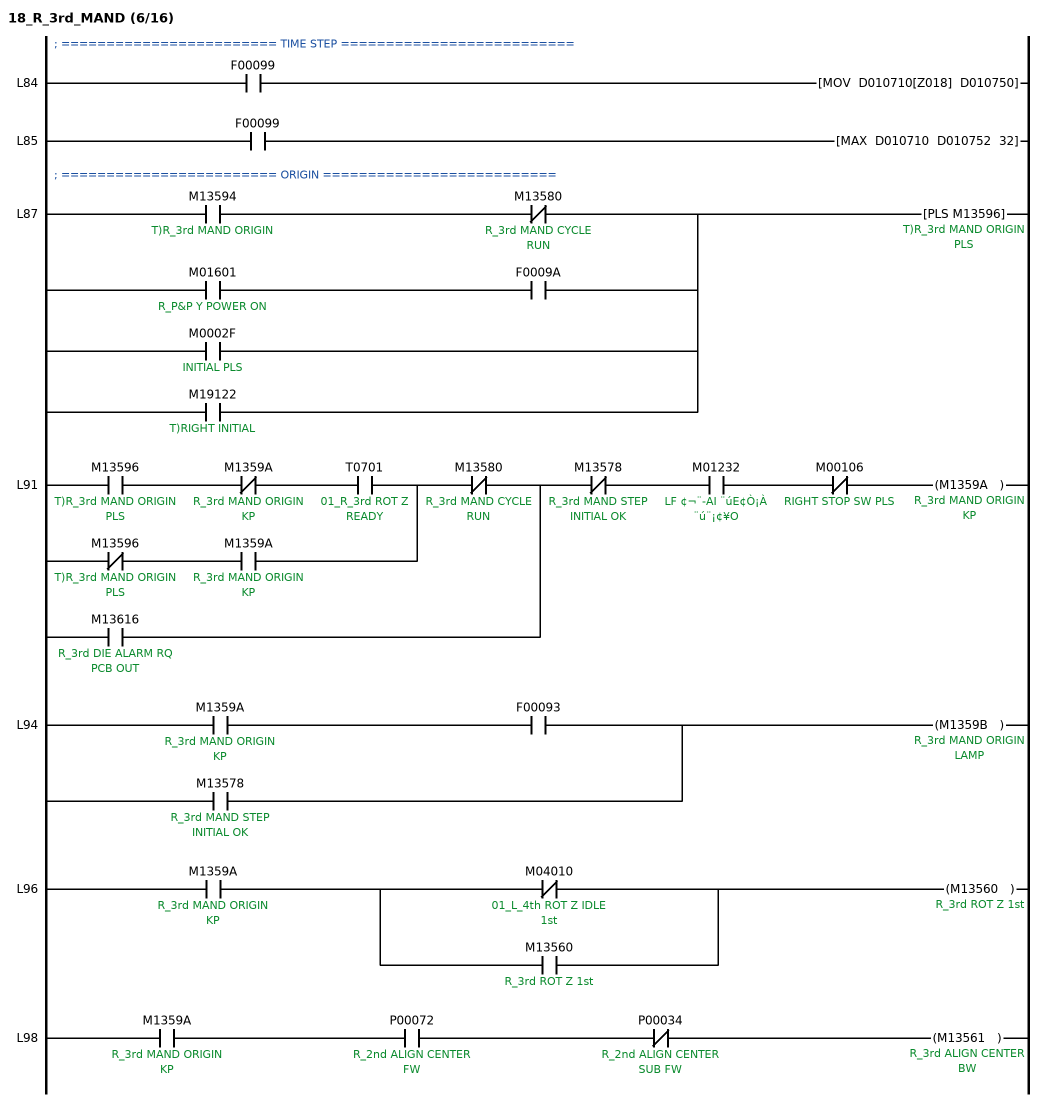
[picture p168: 18_R_3rd_MAND rungs L84-L98]
// ======================== TIME STEP ==========================
; L84
LOAD      F00099
MOV       D010710[Z018] D010750
; L85
LOAD      F00099
MAX       D010710 D010752 32
// ======================== ORIGIN ==========================
; L87
LOAD      M13594	// T)R_3rd MAND ORIGIN
AND NOT   M13580	// R_3rd MAND CYCLE RUN
LOAD      M01601	// R_P&P Y POWER ON
AND       F0009A
OR LOAD
OR        M0002F	// INITIAL PLS
OR        M19122	// T)RIGHT INITIAL
OUTP      M13596	// T)R_3rd MAND ORIGIN PLS
; L91
LOAD      M13596	// T)R_3rd MAND ORIGIN PLS
AND NOT   M1359A	// R_3rd MAND ORIGIN KP
AND       T0701	// 01_R_3rd ROT Z READY
LOAD NOT  M13596	// T)R_3rd MAND ORIGIN PLS
AND       M1359A	// R_3rd MAND ORIGIN KP
OR LOAD
AND NOT   M13580	// R_3rd MAND CYCLE RUN
OR        M13616	// R_3rd DIE ALARM RQ PCB OUT
AND NOT   M13578	// R_3rd MAND STEP INITIAL OK
AND       M01232	// LF ¢¬¨­AI ¨úE¢Ò¡À ¨ú¨¡¢¥O
AND NOT   M00106	// RIGHT STOP SW PLS
OUT       M1359A	// R_3rd MAND ORIGIN KP
; L94
LOAD      M1359A	// R_3rd MAND ORIGIN KP
AND       F00093
OR        M13578	// R_3rd MAND STEP INITIAL OK
OUT       M1359B	// R_3rd MAND ORIGIN LAMP
; L96
LOAD      M1359A	// R_3rd MAND ORIGIN KP
LOAD NOT  M04010	// 01_L_4th ROT Z IDLE 1st
OR        M13560	// R_3rd ROT Z 1st
AND LOAD
OUT       M13560	// R_3rd ROT Z 1st
; L98
LOAD      M1359A	// R_3rd MAND ORIGIN KP
AND       P00072	// R_2nd ALIGN CENTER FW
AND NOT   P00034	// R_2nd ALIGN CENTER SUB FW
OUT       M13561	// R_3rd ALIGN CENTER BW

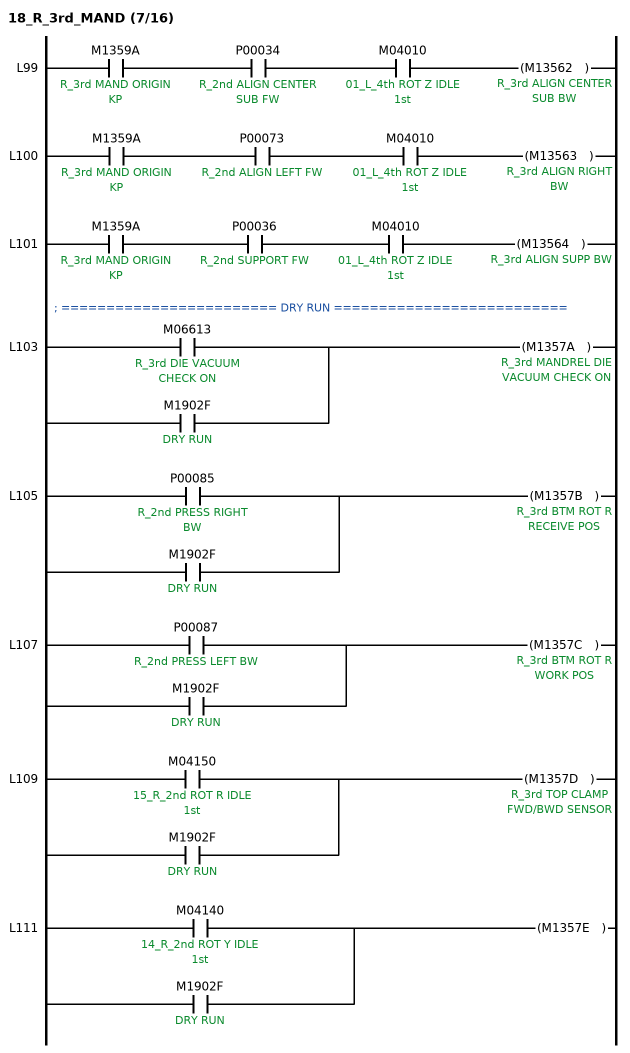
; L99
LOAD      M1359A	// R_3rd MAND ORIGIN KP
AND       P00034	// R_2nd ALIGN CENTER SUB FW
AND       M04010	// 01_L_4th ROT Z IDLE 1st
OUT       M13562	// R_3rd ALIGN CENTER SUB BW
; L100
LOAD      M1359A	// R_3rd MAND ORIGIN KP
AND       P00073	// R_2nd ALIGN LEFT FW
AND       M04010	// 01_L_4th ROT Z IDLE 1st
OUT       M13563	// R_3rd ALIGN RIGHT BW
; L101
LOAD      M1359A	// R_3rd MAND ORIGIN KP
AND       P00036	// R_2nd SUPPORT FW
AND       M04010	// 01_L_4th ROT Z IDLE 1st
OUT       M13564	// R_3rd ALIGN SUPP BW
// ======================== DRY RUN ==========================
; L103
LOAD      M06613	// R_3rd DIE VACUUM CHECK ON
OR        M1902F	// DRY RUN
OUT       M1357A	// R_3rd MANDREL DIE VACUUM CHECK ON
; L105
LOAD      P00085	// R_2nd PRESS RIGHT BW
OR        M1902F	// DRY RUN
OUT       M1357B	// R_3rd BTM ROT R RECEIVE POS
; L107
LOAD      P00087	// R_2nd PRESS LEFT BW
OR        M1902F	// DRY RUN
OUT       M1357C	// R_3rd BTM ROT R WORK POS
; L109
LOAD      M04150	// 15_R_2nd ROT R IDLE 1st
OR        M1902F	// DRY RUN
OUT       M1357D	// R_3rd TOP CLAMP FWD/BWD SENSOR
; L111
LOAD      M04140	// 14_R_2nd ROT Y IDLE 1st
OR        M1902F	// DRY RUN
OUT       M1357E

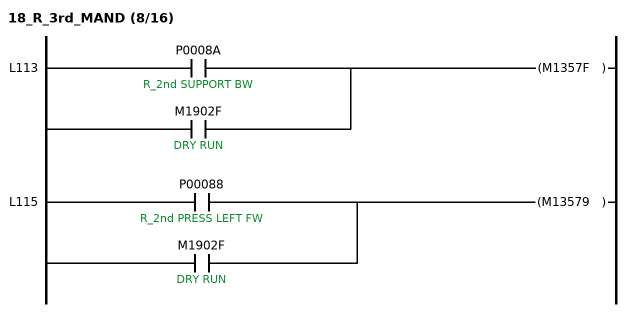
; L113
LOAD      P0008A	// R_2nd SUPPORT BW
OR        M1902F	// DRY RUN
OUT       M1357F
; L115
LOAD      P00088	// R_2nd PRESS LEFT FW
OR        M1902F	// DRY RUN
OUT       M13579

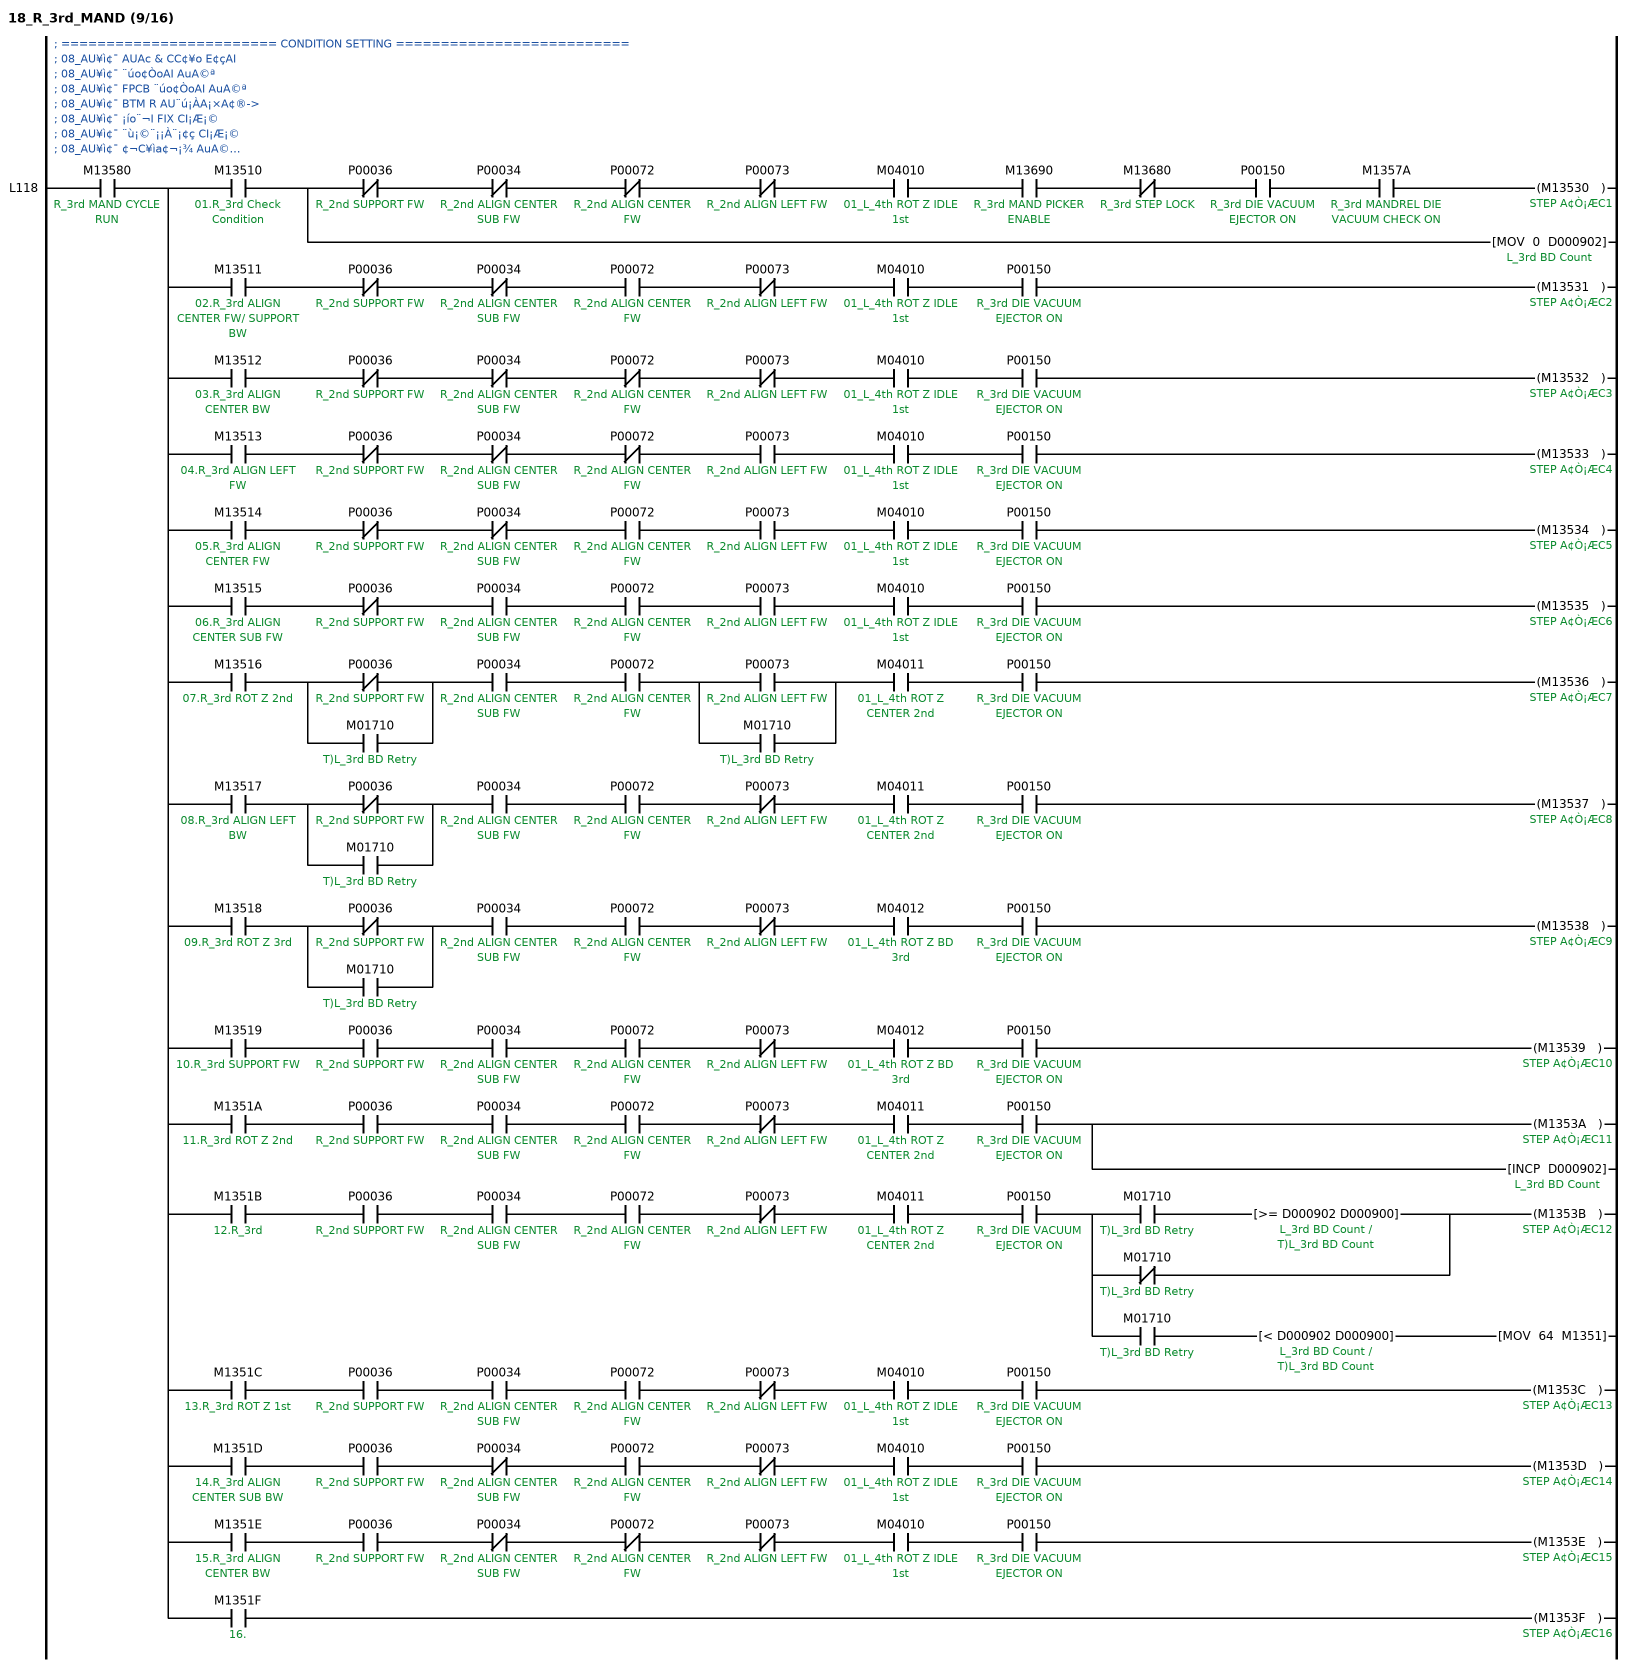
// ======================== CONDITION SETTING ==========================
; L118
LOAD      M13580	// R_3rd MAND CYCLE RUN
MPUSH
AND       M13510	// 01.R_3rd Check Condition
MPUSH
AND NOT   P00036	// R_2nd SUPPORT FW
AND NOT   P00034	// R_2nd ALIGN CENTER SUB FW
AND NOT   P00072	// R_2nd ALIGN CENTER FW
AND NOT   P00073	// R_2nd ALIGN LEFT FW
AND       M04010	// 01_L_4th ROT Z IDLE 1st
AND       M13690	// R_3rd MAND PICKER ENABLE
AND NOT   M13680	// R_3rd STEP LOCK
AND       P00150	// R_3rd DIE VACUUM EJECTOR ON
AND       M1357A	// R_3rd MANDREL DIE VACUUM CHECK ON
OUT       M13530	// STEP A¢Ò¡ÆC1
MPOP
MOV       0 D000902	// L_3rd BD Count
MLOAD
AND       M13511	// 02.R_3rd ALIGN CENTER FW/ SUPPORT BW
AND NOT   P00036	// R_2nd SUPPORT FW
AND NOT   P00034	// R_2nd ALIGN CENTER SUB FW
AND       P00072	// R_2nd ALIGN CENTER FW
AND NOT   P00073	// R_2nd ALIGN LEFT FW
AND       M04010	// 01_L_4th ROT Z IDLE 1st
AND       P00150	// R_3rd DIE VACUUM EJECTOR ON
OUT       M13531	// STEP A¢Ò¡ÆC2
MLOAD
AND       M13512	// 03.R_3rd ALIGN CENTER BW
AND NOT   P00036	// R_2nd SUPPORT FW
AND NOT   P00034	// R_2nd ALIGN CENTER SUB FW
AND NOT   P00072	// R_2nd ALIGN CENTER FW
AND NOT   P00073	// R_2nd ALIGN LEFT FW
AND       M04010	// 01_L_4th ROT Z IDLE 1st
AND       P00150	// R_3rd DIE VACUUM EJECTOR ON
OUT       M13532	// STEP A¢Ò¡ÆC3
MLOAD
AND       M13513	// 04.R_3rd ALIGN LEFT FW
AND NOT   P00036	// R_2nd SUPPORT FW
AND NOT   P00034	// R_2nd ALIGN CENTER SUB FW
AND NOT   P00072	// R_2nd ALIGN CENTER FW
AND       P00073	// R_2nd ALIGN LEFT FW
AND       M04010	// 01_L_4th ROT Z IDLE 1st
AND       P00150	// R_3rd DIE VACUUM EJECTOR ON
OUT       M13533	// STEP A¢Ò¡ÆC4
MLOAD
AND       M13514	// 05.R_3rd ALIGN CENTER FW
AND NOT   P00036	// R_2nd SUPPORT FW
AND NOT   P00034	// R_2nd ALIGN CENTER SUB FW
AND       P00072	// R_2nd ALIGN CENTER FW
AND       P00073	// R_2nd ALIGN LEFT FW
AND       M04010	// 01_L_4th ROT Z IDLE 1st
AND       P00150	// R_3rd DIE VACUUM EJECTOR ON
OUT       M13534	// STEP A¢Ò¡ÆC5
MLOAD
AND       M13515	// 06.R_3rd ALIGN CENTER SUB FW
AND NOT   P00036	// R_2nd SUPPORT FW
AND       P00034	// R_2nd ALIGN CENTER SUB FW
AND       P00072	// R_2nd ALIGN CENTER FW
AND       P00073	// R_2nd ALIGN LEFT FW
AND       M04010	// 01_L_4th ROT Z IDLE 1st
AND       P00150	// R_3rd DIE VACUUM EJECTOR ON
OUT       M13535	// STEP A¢Ò¡ÆC6
MLOAD
AND       M13516	// 07.R_3rd ROT Z 2nd
LOAD NOT  P00036	// R_2nd SUPPORT FW
OR        M01710	// T)L_3rd BD Retry
AND LOAD
AND       P00034	// R_2nd ALIGN CENTER SUB FW
AND       P00072	// R_2nd ALIGN CENTER FW
LOAD      P00073	// R_2nd ALIGN LEFT FW
OR        M01710	// T)L_3rd BD Retry
AND LOAD
AND       M04011	// 01_L_4th ROT Z CENTER 2nd
AND       P00150	// R_3rd DIE VACUUM EJECTOR ON
OUT       M13536	// STEP A¢Ò¡ÆC7
MLOAD
AND       M13517	// 08.R_3rd ALIGN LEFT BW
LOAD NOT  P00036	// R_2nd SUPPORT FW
OR        M01710	// T)L_3rd BD Retry
AND LOAD
AND       P00034	// R_2nd ALIGN CENTER SUB FW
AND       P00072	// R_2nd ALIGN CENTER FW
AND NOT   P00073	// R_2nd ALIGN LEFT FW
AND       M04011	// 01_L_4th ROT Z CENTER 2nd
AND       P00150	// R_3rd DIE VACUUM EJECTOR ON
OUT       M13537	// STEP A¢Ò¡ÆC8
MLOAD
AND       M13518	// 09.R_3rd ROT Z 3rd
LOAD NOT  P00036	// R_2nd SUPPORT FW
OR        M01710	// T)L_3rd BD Retry
AND LOAD
AND       P00034	// R_2nd ALIGN CENTER SUB FW
AND       P00072	// R_2nd ALIGN CENTER FW
AND NOT   P00073	// R_2nd ALIGN LEFT FW
AND       M04012	// 01_L_4th ROT Z BD 3rd
AND       P00150	// R_3rd DIE VACUUM EJECTOR ON
OUT       M13538	// STEP A¢Ò¡ÆC9
MLOAD
AND       M13519	// 10.R_3rd SUPPORT FW
AND       P00036	// R_2nd SUPPORT FW
AND       P00034	// R_2nd ALIGN CENTER SUB FW
AND       P00072	// R_2nd ALIGN CENTER FW
AND NOT   P00073	// R_2nd ALIGN LEFT FW
AND       M04012	// 01_L_4th ROT Z BD 3rd
AND       P00150	// R_3rd DIE VACUUM EJECTOR ON
OUT       M13539	// STEP A¢Ò¡ÆC10
MLOAD
AND       M1351A	// 11.R_3rd ROT Z 2nd
AND       P00036	// R_2nd SUPPORT FW
AND       P00034	// R_2nd ALIGN CENTER SUB FW
AND       P00072	// R_2nd ALIGN CENTER FW
AND NOT   P00073	// R_2nd ALIGN LEFT FW
AND       M04011	// 01_L_4th ROT Z CENTER 2nd
AND       P00150	// R_3rd DIE VACUUM EJECTOR ON
OUT       M1353A	// STEP A¢Ò¡ÆC11
INCP      D000902	// L_3rd BD Count
MLOAD
AND       M1351B	// 12.R_3rd 
AND       P00036	// R_2nd SUPPORT FW
AND       P00034	// R_2nd ALIGN CENTER SUB FW
AND       P00072	// R_2nd ALIGN CENTER FW
AND NOT   P00073	// R_2nd ALIGN LEFT FW
AND       M04011	// 01_L_4th ROT Z CENTER 2nd
AND       P00150	// R_3rd DIE VACUUM EJECTOR ON
MPUSH
LOAD      M01710	// T)L_3rd BD Retry
AND>=     D000902 D000900	// L_3rd BD Count / T)L_3rd BD Count
OR NOT    M01710	// T)L_3rd BD Retry
AND LOAD
OUT       M1353B	// STEP A¢Ò¡ÆC12
MPOP
AND       M01710	// T)L_3rd BD Retry
AND<      D000902 D000900	// L_3rd BD Count / T)L_3rd BD Count
MOV       64 M1351
MLOAD
AND       M1351C	// 13.R_3rd ROT Z 1st
AND       P00036	// R_2nd SUPPORT FW
AND       P00034	// R_2nd ALIGN CENTER SUB FW
AND       P00072	// R_2nd ALIGN CENTER FW
AND NOT   P00073	// R_2nd ALIGN LEFT FW
AND       M04010	// 01_L_4th ROT Z IDLE 1st
AND       P00150	// R_3rd DIE VACUUM EJECTOR ON
OUT       M1353C	// STEP A¢Ò¡ÆC13
MLOAD
AND       M1351D	// 14.R_3rd ALIGN CENTER SUB BW
AND       P00036	// R_2nd SUPPORT FW
AND NOT   P00034	// R_2nd ALIGN CENTER SUB FW
AND       P00072	// R_2nd ALIGN CENTER FW
AND NOT   P00073	// R_2nd ALIGN LEFT FW
AND       M04010	// 01_L_4th ROT Z IDLE 1st
AND       P00150	// R_3rd DIE VACUUM EJECTOR ON
OUT       M1353D	// STEP A¢Ò¡ÆC14
MLOAD
AND       M1351E	// 15.R_3rd ALIGN CENTER BW
AND       P00036	// R_2nd SUPPORT FW
AND NOT   P00034	// R_2nd ALIGN CENTER SUB FW
AND NOT   P00072	// R_2nd ALIGN CENTER FW
AND NOT   P00073	// R_2nd ALIGN LEFT FW
AND       M04010	// 01_L_4th ROT Z IDLE 1st
AND       P00150	// R_3rd DIE VACUUM EJECTOR ON
OUT       M1353E	// STEP A¢Ò¡ÆC15
MPOP
AND       M1351F	// 16.
OUT       M1353F	// STEP A¢Ò¡ÆC16
// output comment: 08_AU¥ì¢¯ AUAc & CC¢¥o E¢çAI
// output comment: 08_AU¥ì¢¯ ¨úo¢ÒoAI AuA©ª
// output comment: 08_AU¥ì¢¯ FPCB ¨úo¢ÒoAI AuA©ª
// output comment: 08_AU¥ì¢¯ BTM R AU¨ú¡ÀA¡×A¢®->
// output comment: 08_AU¥ì¢¯ ¡ío¨¬I FIX CI¡Æ¡©
// output comment: 08_AU¥ì¢¯ ¨ù¡©¨¡¡À¨¡¢ç CI¡Æ¡©
// output comment: 08_AU¥ì¢¯ ¢¬C¥ìa¢¬¡¾ AuA©ª
// output comment: 08_AU¥ì¢¯ ¢¬C¥ìa¢¬¡¾ E¢¬Au
// output comment: 08_AU¥ì¢¯ ¢¬C¥ìa¢¬¡¾ ¨¬©ö¡¾I

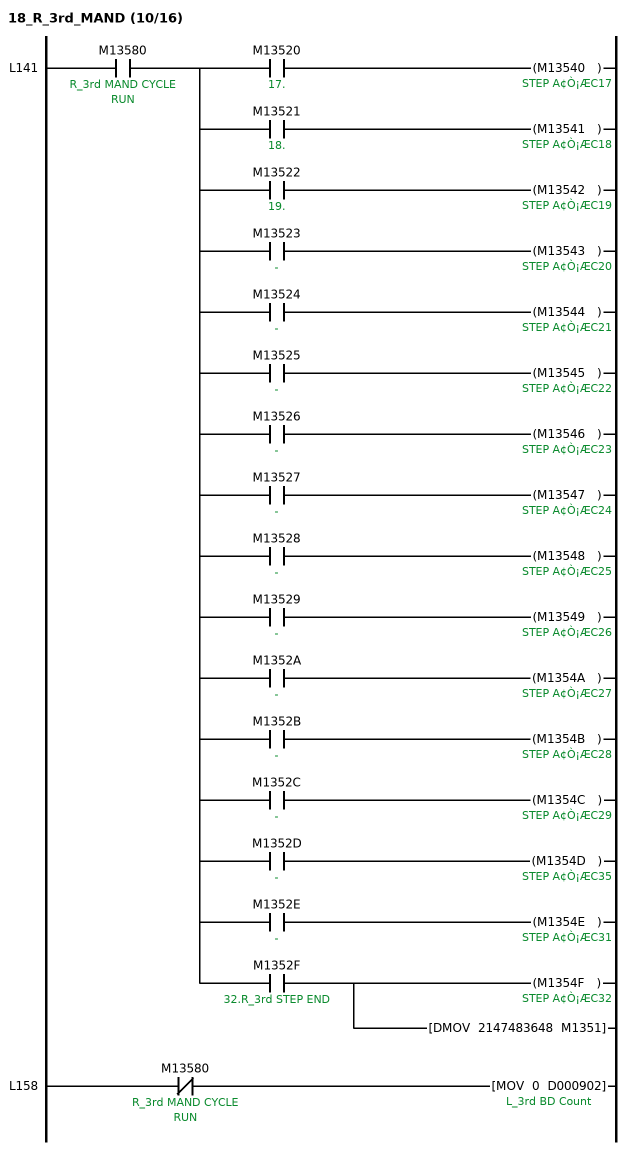
; L141
LOAD      M13580	// R_3rd MAND CYCLE RUN
MPUSH
AND       M13520	// 17.
OUT       M13540	// STEP A¢Ò¡ÆC17
MLOAD
AND       M13521	// 18.
OUT       M13541	// STEP A¢Ò¡ÆC18
MLOAD
AND       M13522	// 19.
OUT       M13542	// STEP A¢Ò¡ÆC19
MLOAD
AND       M13523	// -
OUT       M13543	// STEP A¢Ò¡ÆC20
MLOAD
AND       M13524	// -
OUT       M13544	// STEP A¢Ò¡ÆC21
MLOAD
AND       M13525	// -
OUT       M13545	// STEP A¢Ò¡ÆC22
MLOAD
AND       M13526	// -
OUT       M13546	// STEP A¢Ò¡ÆC23
MLOAD
AND       M13527	// -
OUT       M13547	// STEP A¢Ò¡ÆC24
MLOAD
AND       M13528	// -
OUT       M13548	// STEP A¢Ò¡ÆC25
MLOAD
AND       M13529	// -
OUT       M13549	// STEP A¢Ò¡ÆC26
MLOAD
AND       M1352A	// -
OUT       M1354A	// STEP A¢Ò¡ÆC27
MLOAD
AND       M1352B	// -
OUT       M1354B	// STEP A¢Ò¡ÆC28
MLOAD
AND       M1352C	// -
OUT       M1354C	// STEP A¢Ò¡ÆC29
MLOAD
AND       M1352D	// -
OUT       M1354D	// STEP A¢Ò¡ÆC35
MLOAD
AND       M1352E	// -
OUT       M1354E	// STEP A¢Ò¡ÆC31
MPOP
AND       M1352F	// 32.R_3rd STEP END
OUT       M1354F	// STEP A¢Ò¡ÆC32
DMOV      2147483648 M1351
; L158
LOAD NOT  M13580	// R_3rd MAND CYCLE RUN
MOV       0 D000902	// L_3rd BD Count

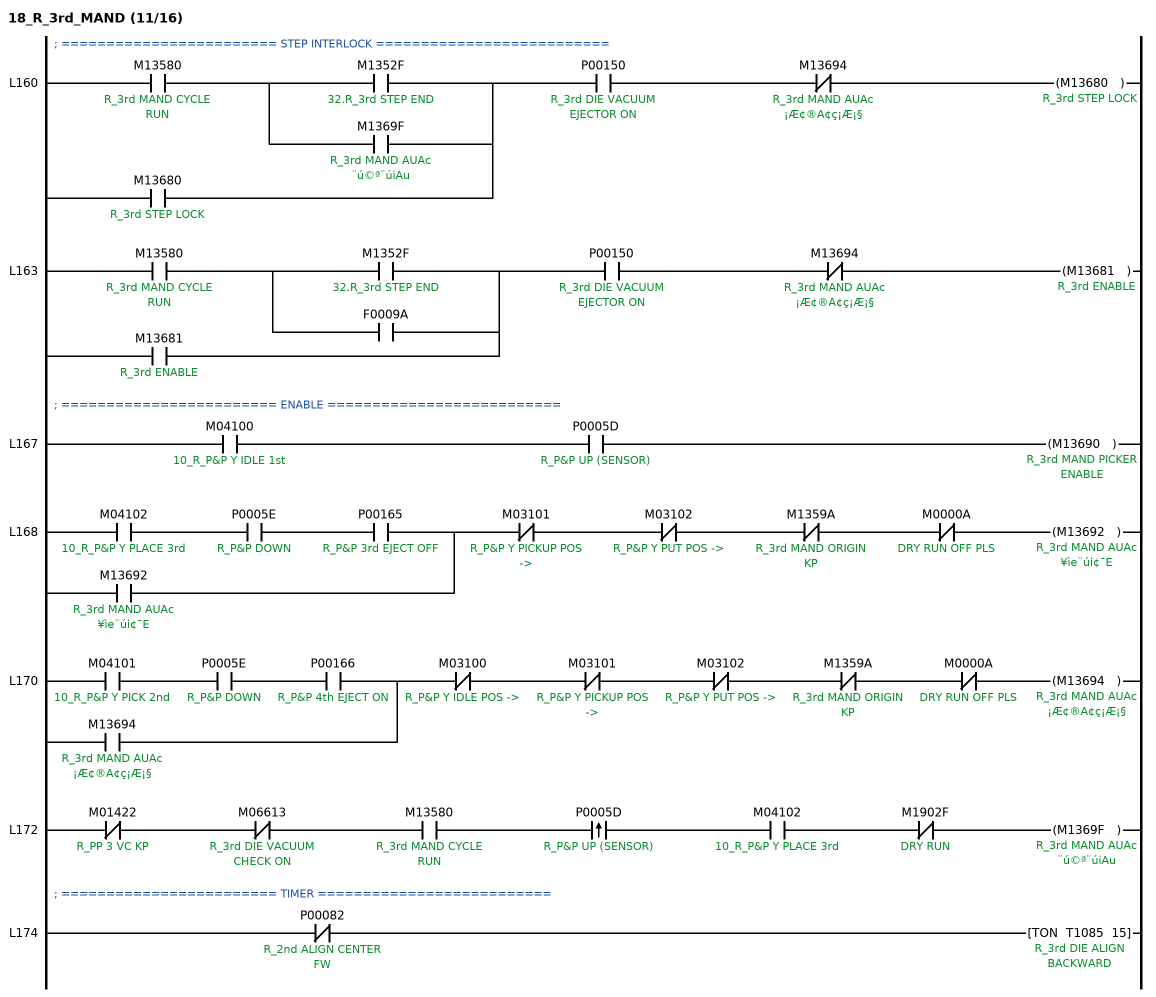
// ======================== STEP INTERLOCK ==========================
; L160
LOAD      M13580	// R_3rd MAND CYCLE RUN
LOAD      M1352F	// 32.R_3rd STEP END
OR        M1369F	// R_3rd MAND AUAc ¨ú©ª¨úiAu
AND LOAD
OR        M13680	// R_3rd STEP LOCK
AND       P00150	// R_3rd DIE VACUUM EJECTOR ON
AND NOT   M13694	// R_3rd MAND AUAc ¡Æ¢®A¢ç¡Æ¡§
OUT       M13680	// R_3rd STEP LOCK
; L163
LOAD      M13580	// R_3rd MAND CYCLE RUN
LOAD      M1352F	// 32.R_3rd STEP END
OR        F0009A
AND LOAD
OR        M13681	// R_3rd ENABLE
AND       P00150	// R_3rd DIE VACUUM EJECTOR ON
AND NOT   M13694	// R_3rd MAND AUAc ¡Æ¢®A¢ç¡Æ¡§
OUT       M13681	// R_3rd ENABLE
// ======================== ENABLE ==========================
; L167
LOAD      M04100	// 10_R_P&P Y IDLE 1st
AND       P0005D	// R_P&P UP (SENSOR)
OUT       M13690	// R_3rd MAND PICKER ENABLE
; L168
LOAD      M04102	// 10_R_P&P Y PLACE 3rd
AND       P0005E	// R_P&P DOWN
AND       P00165	// R_P&P 3rd EJECT OFF
OR        M13692	// R_3rd MAND AUAc ¥ìe¨úi¢¯E
AND NOT   M03101	// R_P&P Y PICKUP POS ->
AND NOT   M03102	// R_P&P Y PUT POS ->
AND NOT   M1359A	// R_3rd MAND ORIGIN KP
AND NOT   M0000A	// DRY RUN OFF PLS
OUT       M13692	// R_3rd MAND AUAc ¥ìe¨úi¢¯E
; L170
LOAD      M04101	// 10_R_P&P Y PICK 2nd
AND       P0005E	// R_P&P DOWN
AND       P00166	// R_P&P 4th EJECT ON
OR        M13694	// R_3rd MAND AUAc ¡Æ¢®A¢ç¡Æ¡§
AND NOT   M03100	// R_P&P Y IDLE POS ->
AND NOT   M03101	// R_P&P Y PICKUP POS ->
AND NOT   M03102	// R_P&P Y PUT POS ->
AND NOT   M1359A	// R_3rd MAND ORIGIN KP
AND NOT   M0000A	// DRY RUN OFF PLS
OUT       M13694	// R_3rd MAND AUAc ¡Æ¢®A¢ç¡Æ¡§
; L172
LOAD NOT  M01422	// R_PP 3 VC KP
AND NOT   M06613	// R_3rd DIE VACUUM CHECK ON
AND       M13580	// R_3rd MAND CYCLE RUN
ANDP      P0005D	// R_P&P UP (SENSOR)
AND       M04102	// 10_R_P&P Y PLACE 3rd
AND NOT   M1902F	// DRY RUN
OUT       M1369F	// R_3rd MAND AUAc ¨ú©ª¨úiAu
// ======================== TIMER ==========================
; L174
LOAD NOT  P00082	// R_2nd ALIGN CENTER FW
TON       T1085 15	// R_3rd DIE ALIGN BACKWARD

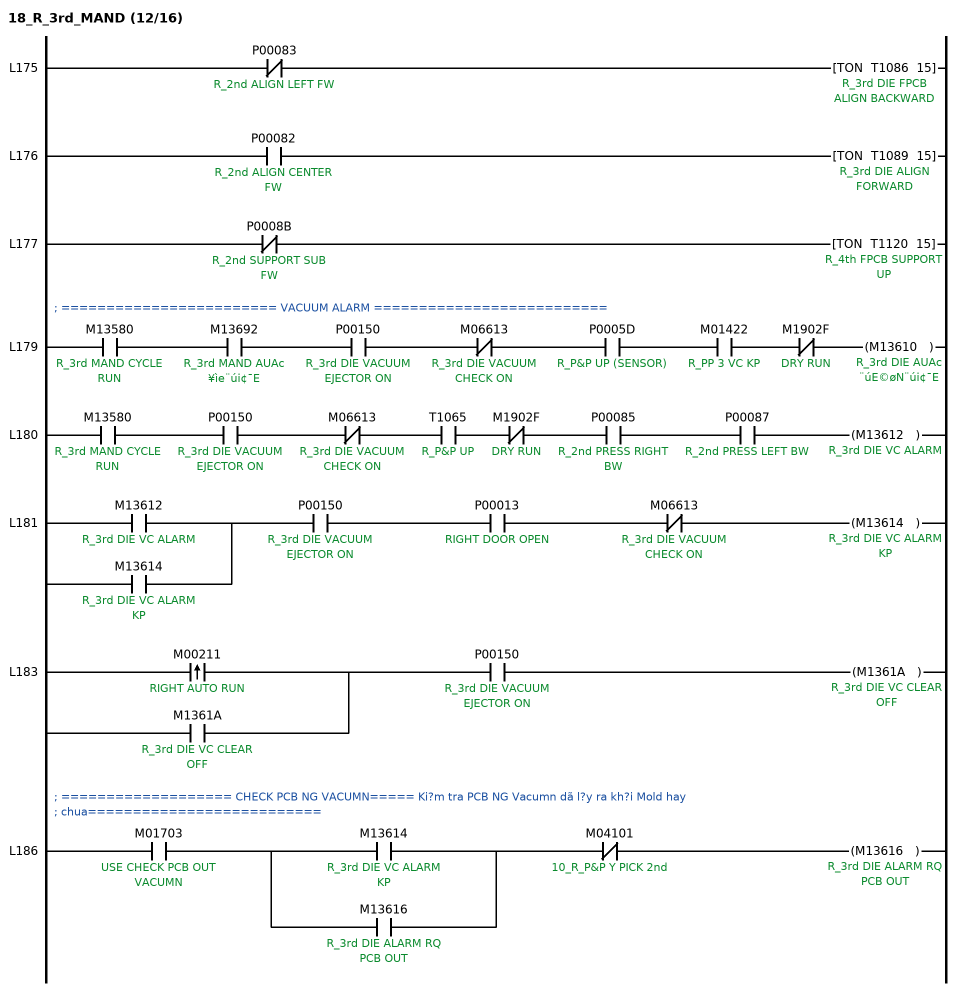
; L175
LOAD NOT  P00083	// R_2nd ALIGN LEFT FW
TON       T1086 15	// R_3rd DIE FPCB ALIGN BACKWARD
; L176
LOAD      P00082	// R_2nd ALIGN CENTER FW
TON       T1089 15	// R_3rd DIE ALIGN FORWARD
; L177
LOAD NOT  P0008B	// R_2nd SUPPORT SUB FW
TON       T1120 15	// R_4th FPCB SUPPORT UP
// ======================== VACUUM ALARM ==========================
; L179
LOAD      M13580	// R_3rd MAND CYCLE RUN
AND       M13692	// R_3rd MAND AUAc ¥ìe¨úi¢¯E
AND       P00150	// R_3rd DIE VACUUM EJECTOR ON
AND NOT   M06613	// R_3rd DIE VACUUM CHECK ON
AND       P0005D	// R_P&P UP (SENSOR)
AND       M01422	// R_PP 3 VC KP
AND NOT   M1902F	// DRY RUN
OUT       M13610	// R_3rd DIE AUAc ¨úE©øN¨úi¢¯E
; L180
LOAD      M13580	// R_3rd MAND CYCLE RUN
AND       P00150	// R_3rd DIE VACUUM EJECTOR ON
AND NOT   M06613	// R_3rd DIE VACUUM CHECK ON
AND       T1065	// R_P&P UP
AND NOT   M1902F	// DRY RUN
AND       P00085	// R_2nd PRESS RIGHT BW
AND       P00087	// R_2nd PRESS LEFT BW
OUT       M13612	// R_3rd DIE VC ALARM
; L181
LOAD      M13612	// R_3rd DIE VC ALARM
OR        M13614	// R_3rd DIE VC ALARM KP
AND       P00150	// R_3rd DIE VACUUM EJECTOR ON
AND       P00013	// RIGHT DOOR OPEN
AND NOT   M06613	// R_3rd DIE VACUUM CHECK ON
OUT       M13614	// R_3rd DIE VC ALARM KP
; L183
LOADP     M00211	// RIGHT AUTO RUN
OR        M1361A	// R_3rd DIE VC CLEAR OFF
AND       P00150	// R_3rd DIE VACUUM EJECTOR ON
OUT       M1361A	// R_3rd DIE VC CLEAR OFF
// =================== CHECK PCB NG VACUMN===== Ki?m tra PCB NG Vacumn dã l?y ra kh?i Mold hay chua==========================
; L186
LOAD      M01703	// USE CHECK PCB OUT VACUMN
LOAD      M13614	// R_3rd DIE VC ALARM KP
OR        M13616	// R_3rd DIE ALARM RQ PCB OUT
AND LOAD
AND NOT   M04101	// 10_R_P&P Y PICK 2nd
OUT       M13616	// R_3rd DIE ALARM RQ PCB OUT

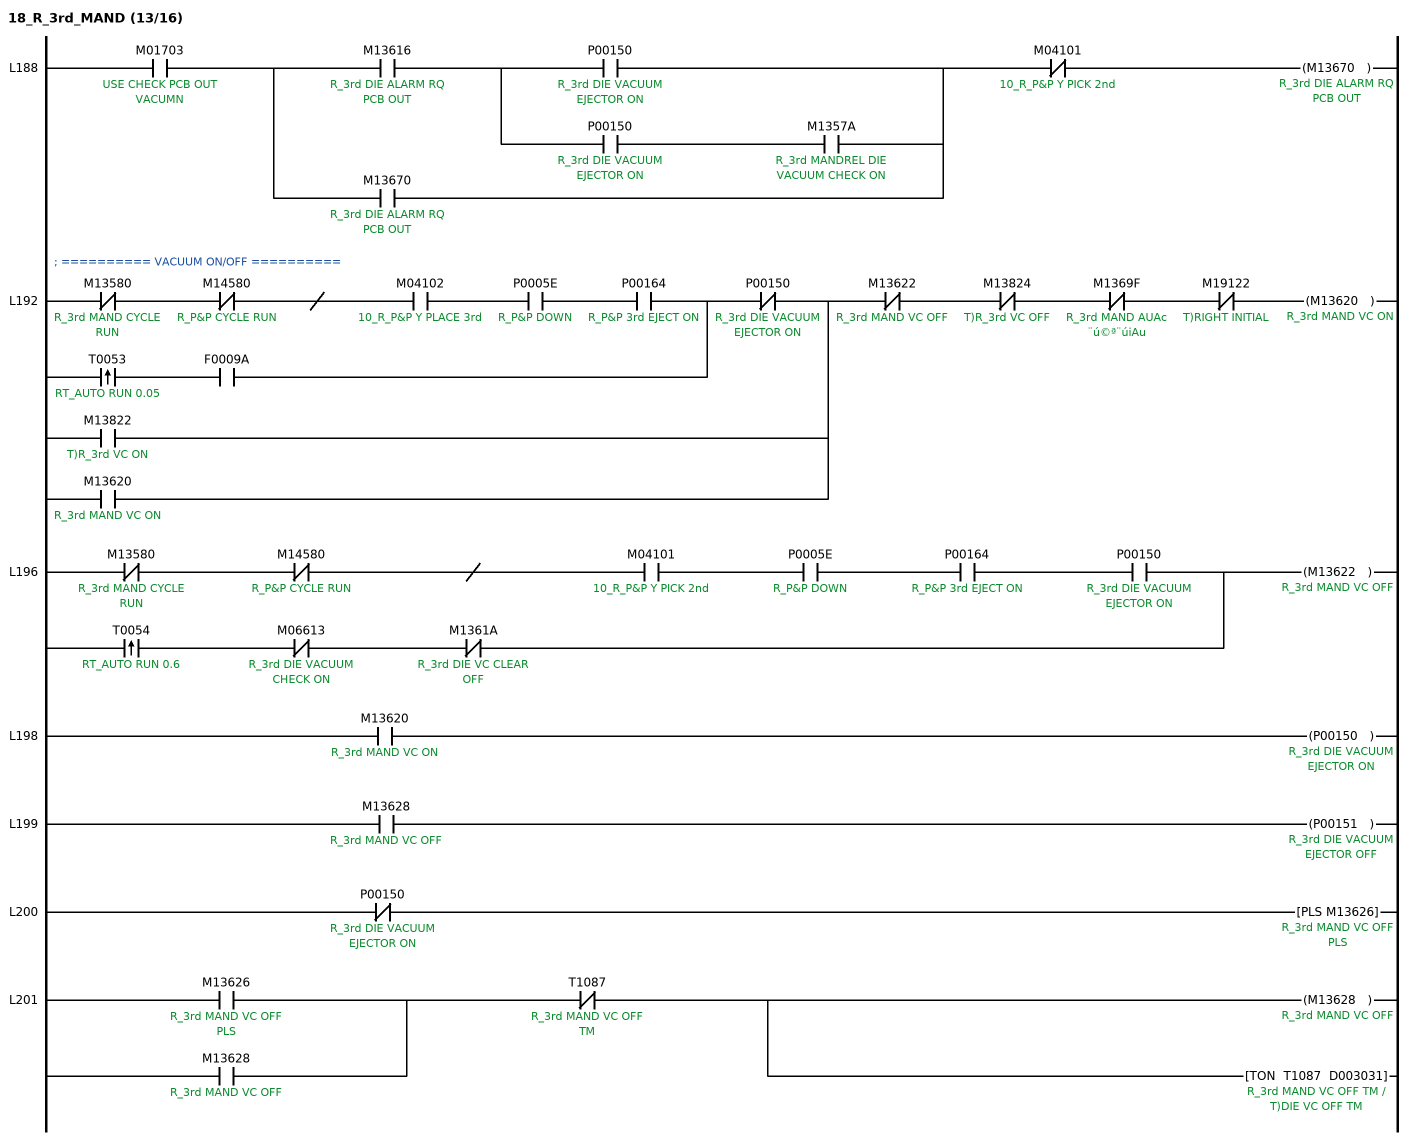
; L188
LOAD      M01703	// USE CHECK PCB OUT VACUMN
LOAD      M13616	// R_3rd DIE ALARM RQ PCB OUT
LOAD      P00150	// R_3rd DIE VACUUM EJECTOR ON
LOAD      P00150	// R_3rd DIE VACUUM EJECTOR ON
AND       M1357A	// R_3rd MANDREL DIE VACUUM CHECK ON
OR LOAD
AND LOAD
OR        M13670	// R_3rd DIE ALARM RQ PCB OUT
AND LOAD
AND NOT   M04101	// 10_R_P&P Y PICK 2nd
OUT       M13670	// R_3rd DIE ALARM RQ PCB OUT
// ========== VACUUM ON/OFF ==========
; L192
LOAD NOT  M13580	// R_3rd MAND CYCLE RUN
AND NOT   M14580	// R_P&P CYCLE RUN
NOT
AND       M04102	// 10_R_P&P Y PLACE 3rd
AND       P0005E	// R_P&P DOWN
AND       P00164	// R_P&P 3rd EJECT ON
LOADP     T0053	// RT_AUTO RUN 0.05
AND       F0009A
OR LOAD
AND NOT   P00150	// R_3rd DIE VACUUM EJECTOR ON
OR        M13822	// T)R_3rd VC ON
OR        M13620	// R_3rd MAND VC ON
AND NOT   M13622	// R_3rd MAND VC OFF
AND NOT   M13824	// T)R_3rd VC OFF
AND NOT   M1369F	// R_3rd MAND AUAc ¨ú©ª¨úiAu
AND NOT   M19122	// T)RIGHT INITIAL
OUT       M13620	// R_3rd MAND VC ON
; L196
LOAD NOT  M13580	// R_3rd MAND CYCLE RUN
AND NOT   M14580	// R_P&P CYCLE RUN
NOT
AND       M04101	// 10_R_P&P Y PICK 2nd
AND       P0005E	// R_P&P DOWN
AND       P00164	// R_P&P 3rd EJECT ON
AND       P00150	// R_3rd DIE VACUUM EJECTOR ON
LOADP     T0054	// RT_AUTO RUN 0.6
AND NOT   M06613	// R_3rd DIE VACUUM CHECK ON
AND NOT   M1361A	// R_3rd DIE VC CLEAR OFF
OR LOAD
OUT       M13622	// R_3rd MAND VC OFF
; L198
LOAD      M13620	// R_3rd MAND VC ON
OUT       P00150	// R_3rd DIE VACUUM EJECTOR ON
; L199
LOAD      M13628	// R_3rd MAND VC OFF
OUT       P00151	// R_3rd DIE VACUUM EJECTOR OFF
; L200
LOAD NOT  P00150	// R_3rd DIE VACUUM EJECTOR ON
OUTP      M13626	// R_3rd MAND VC OFF PLS
; L201
LOAD      M13626	// R_3rd MAND VC OFF PLS
OR        M13628	// R_3rd MAND VC OFF
AND NOT   T1087	// R_3rd MAND VC OFF TM
OUT       M13628	// R_3rd MAND VC OFF
TON       T1087 D003031	// R_3rd MAND VC OFF TM / T)DIE VC OFF TM

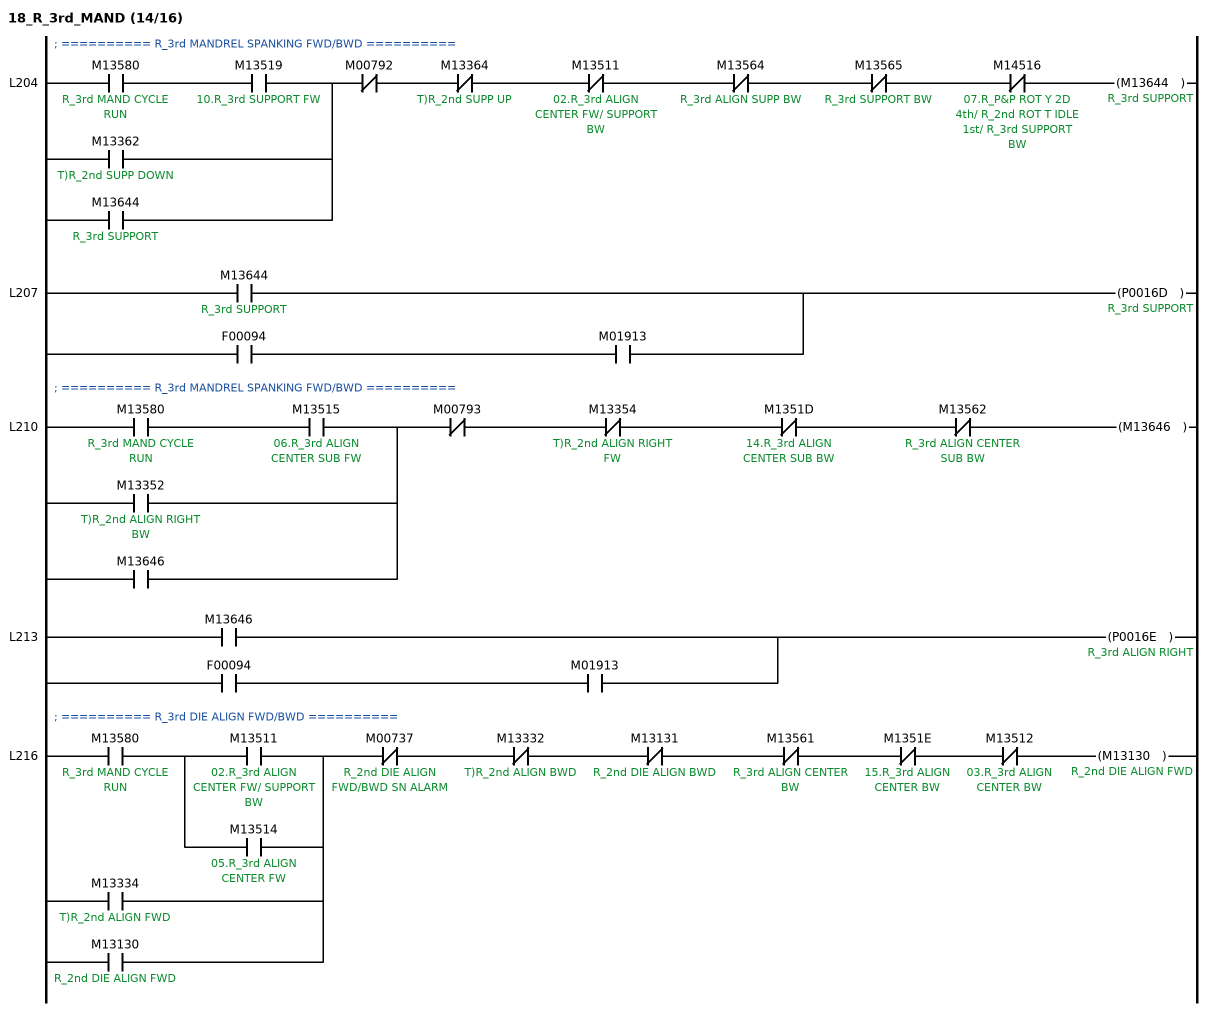
// ========== R_3rd MANDREL SPANKING FWD/BWD ==========
; L204
LOAD      M13580	// R_3rd MAND CYCLE RUN
AND       M13519	// 10.R_3rd SUPPORT FW
OR        M13362	// T)R_2nd SUPP DOWN
OR        M13644	// R_3rd SUPPORT
AND NOT   M00792
AND NOT   M13364	// T)R_2nd SUPP UP
AND NOT   M13511	// 02.R_3rd ALIGN CENTER FW/ SUPPORT BW
AND NOT   M13564	// R_3rd ALIGN SUPP BW
AND NOT   M13565	// R_3rd SUPPORT BW
AND NOT   M14516	// 07.R_P&P ROT Y 2D 4th/ R_2nd ROT T IDLE 1st/ R_3rd SUPPORT BW
OUT       M13644	// R_3rd SUPPORT
; L207
LOAD      M13644	// R_3rd SUPPORT
LOAD      F00094
AND       M01913
OR LOAD
OUT       P0016D	// R_3rd SUPPORT
// ========== R_3rd MANDREL SPANKING FWD/BWD ==========
; L210
LOAD      M13580	// R_3rd MAND CYCLE RUN
AND       M13515	// 06.R_3rd ALIGN CENTER SUB FW
OR        M13352	// T)R_2nd ALIGN RIGHT BW
OR        M13646
AND NOT   M00793
AND NOT   M13354	// T)R_2nd ALIGN RIGHT FW
AND NOT   M1351D	// 14.R_3rd ALIGN CENTER SUB BW
AND NOT   M13562	// R_3rd ALIGN CENTER SUB BW
OUT       M13646
; L213
LOAD      M13646
LOAD      F00094
AND       M01913
OR LOAD
OUT       P0016E	// R_3rd ALIGN RIGHT
// ========== R_3rd DIE ALIGN FWD/BWD ==========
; L216
LOAD      M13580	// R_3rd MAND CYCLE RUN
LOAD      M13511	// 02.R_3rd ALIGN CENTER FW/ SUPPORT BW
OR        M13514	// 05.R_3rd ALIGN CENTER FW
AND LOAD
OR        M13334	// T)R_2nd ALIGN FWD
OR        M13130	// R_2nd DIE ALIGN FWD
AND NOT   M00737	// R_2nd DIE ALIGN FWD/BWD SN ALARM
AND NOT   M13332	// T)R_2nd ALIGN BWD
AND NOT   M13131	// R_2nd DIE ALIGN BWD
AND NOT   M13561	// R_3rd ALIGN CENTER BW
AND NOT   M1351E	// 15.R_3rd ALIGN CENTER BW
AND NOT   M13512	// 03.R_3rd ALIGN CENTER BW
OUT       M13130	// R_2nd DIE ALIGN FWD

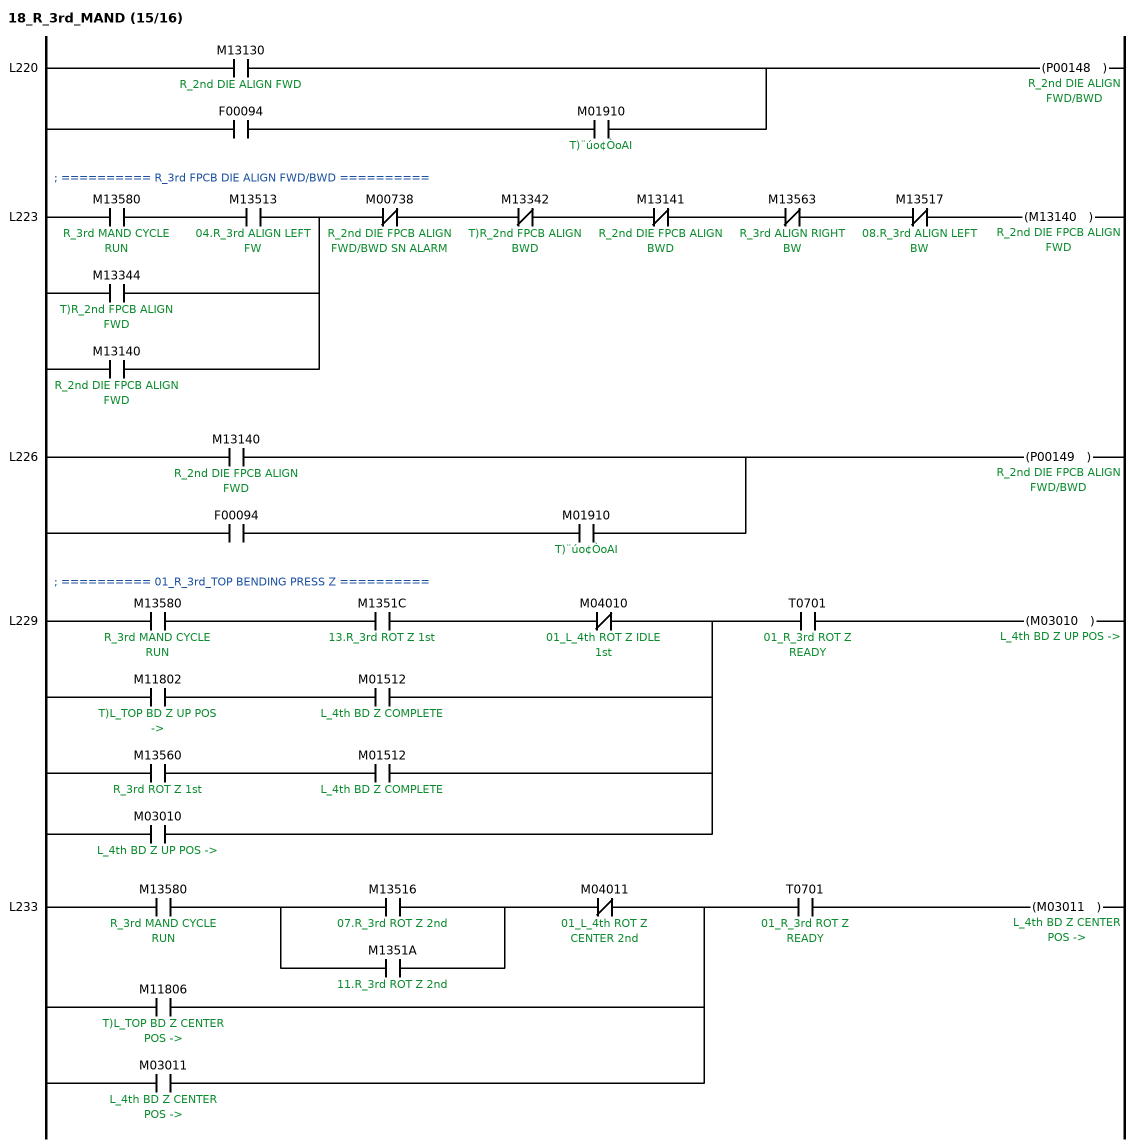
; L220
LOAD      M13130	// R_2nd DIE ALIGN FWD
LOAD      F00094
AND       M01910	// T)¨úo¢ÒoAI
OR LOAD
OUT       P00148	// R_2nd DIE ALIGN FWD/BWD
// ========== R_3rd FPCB DIE ALIGN FWD/BWD ==========
; L223
LOAD      M13580	// R_3rd MAND CYCLE RUN
AND       M13513	// 04.R_3rd ALIGN LEFT FW
OR        M13344	// T)R_2nd FPCB ALIGN FWD
OR        M13140	// R_2nd DIE FPCB ALIGN FWD
AND NOT   M00738	// R_2nd DIE FPCB ALIGN FWD/BWD SN ALARM
AND NOT   M13342	// T)R_2nd FPCB ALIGN BWD
AND NOT   M13141	// R_2nd DIE FPCB ALIGN BWD
AND NOT   M13563	// R_3rd ALIGN RIGHT BW
AND NOT   M13517	// 08.R_3rd ALIGN LEFT BW
OUT       M13140	// R_2nd DIE FPCB ALIGN FWD
; L226
LOAD      M13140	// R_2nd DIE FPCB ALIGN FWD
LOAD      F00094
AND       M01910	// T)¨úo¢ÒoAI
OR LOAD
OUT       P00149	// R_2nd DIE FPCB ALIGN FWD/BWD
// ========== 01_R_3rd_TOP BENDING PRESS Z ==========
; L229
LOAD      M13580	// R_3rd MAND CYCLE RUN
AND       M1351C	// 13.R_3rd ROT Z 1st
AND NOT   M04010	// 01_L_4th ROT Z IDLE 1st
LOAD      M11802	// T)L_TOP BD Z UP POS ->
AND       M01512	// L_4th BD Z COMPLETE
OR LOAD
LOAD      M13560	// R_3rd ROT Z 1st
AND       M01512	// L_4th BD Z COMPLETE
OR LOAD
OR        M03010	// L_4th BD Z UP POS ->
AND       T0701	// 01_R_3rd ROT Z READY
OUT       M03010	// L_4th BD Z UP POS ->
; L233
LOAD      M13580	// R_3rd MAND CYCLE RUN
LOAD      M13516	// 07.R_3rd ROT Z 2nd
OR        M1351A	// 11.R_3rd ROT Z 2nd
AND LOAD
AND NOT   M04011	// 01_L_4th ROT Z CENTER 2nd
OR        M11806	// T)L_TOP BD Z CENTER POS ->
OR        M03011	// L_4th BD Z CENTER POS ->
AND       T0701	// 01_R_3rd ROT Z READY
OUT       M03011	// L_4th BD Z CENTER POS ->

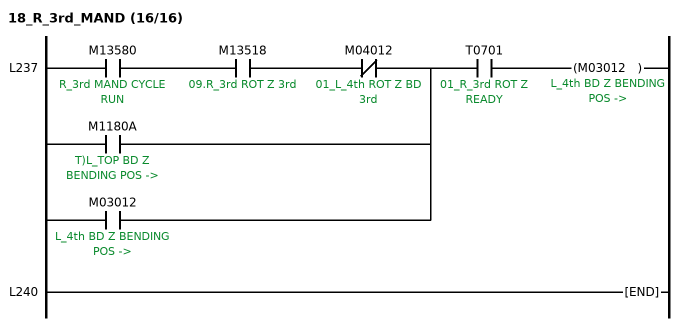
; L237
LOAD      M13580	// R_3rd MAND CYCLE RUN
AND       M13518	// 09.R_3rd ROT Z 3rd
AND NOT   M04012	// 01_L_4th ROT Z BD 3rd
OR        M1180A	// T)L_TOP BD Z BENDING POS ->
OR        M03012	// L_4th BD Z BENDING POS ->
AND       T0701	// 01_R_3rd ROT Z READY
OUT       M03012	// L_4th BD Z BENDING POS ->
; L240
END

PROGRAM 19_R_TOOL (task: ¨ö¨¬A¥ì CA¡¤I¡¾¡¿¡¤¡Í)

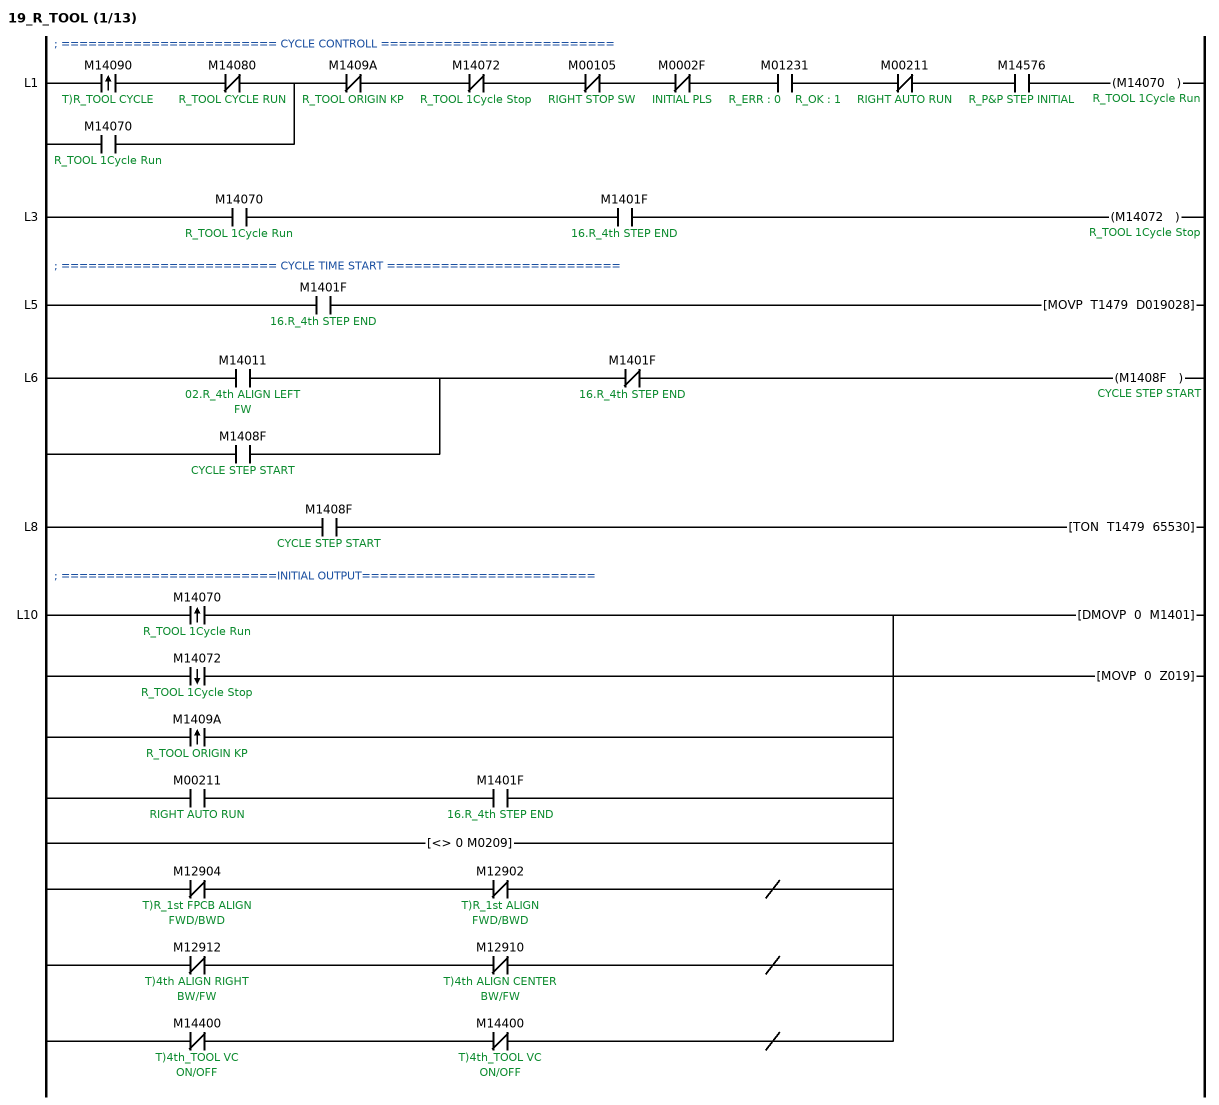
// ======================== CYCLE CONTROLL ==========================
; L1
LOADP     M14090	// T)R_TOOL CYCLE
AND NOT   M14080	// R_TOOL CYCLE RUN
OR        M14070	// R_TOOL 1Cycle Run
AND NOT   M1409A	// R_TOOL ORIGIN KP
AND NOT   M14072	// R_TOOL 1Cycle Stop
AND NOT   M00105	// RIGHT STOP SW
AND NOT   M0002F	// INITIAL PLS
AND       M01231	// R_ERR : 0    R_OK : 1
AND NOT   M00211	// RIGHT AUTO RUN
AND       M14576	// R_P&P STEP INITIAL
OUT       M14070	// R_TOOL 1Cycle Run
; L3
LOAD      M14070	// R_TOOL 1Cycle Run
AND       M1401F	// 16.R_4th STEP END
OUT       M14072	// R_TOOL 1Cycle Stop
// ======================== CYCLE TIME START ==========================
; L5
LOAD      M1401F	// 16.R_4th STEP END
MOVP      T1479 D019028
; L6
LOAD      M14011	// 02.R_4th ALIGN LEFT FW
OR        M1408F	// CYCLE STEP START
AND NOT   M1401F	// 16.R_4th STEP END
OUT       M1408F	// CYCLE STEP START
; L8
LOAD      M1408F	// CYCLE STEP START
TON       T1479 65530
// ========================INITIAL OUTPUT==========================
; L10
LOADP     M14070	// R_TOOL 1Cycle Run
ORN       M14072	// R_TOOL 1Cycle Stop
ORP       M1409A	// R_TOOL ORIGIN KP
LOAD      M00211	// RIGHT AUTO RUN
AND       M1401F	// 16.R_4th STEP END
OR LOAD
OR<>      0 M0209
LOAD NOT  M12904	// T)R_1st FPCB ALIGN FWD/BWD
AND NOT   M12902	// T)R_1st ALIGN FWD/BWD
NOT
OR LOAD
LOAD NOT  M12912	// T)4th ALIGN RIGHT BW/FW
AND NOT   M12910	// T)4th ALIGN CENTER BW/FW
NOT
OR LOAD
LOAD NOT  M14400	// T)4th_TOOL VC ON/OFF
AND NOT   M14400	// T)4th_TOOL VC ON/OFF
NOT
OR LOAD
DMOVP     0 M1401
MOVP      0 Z019

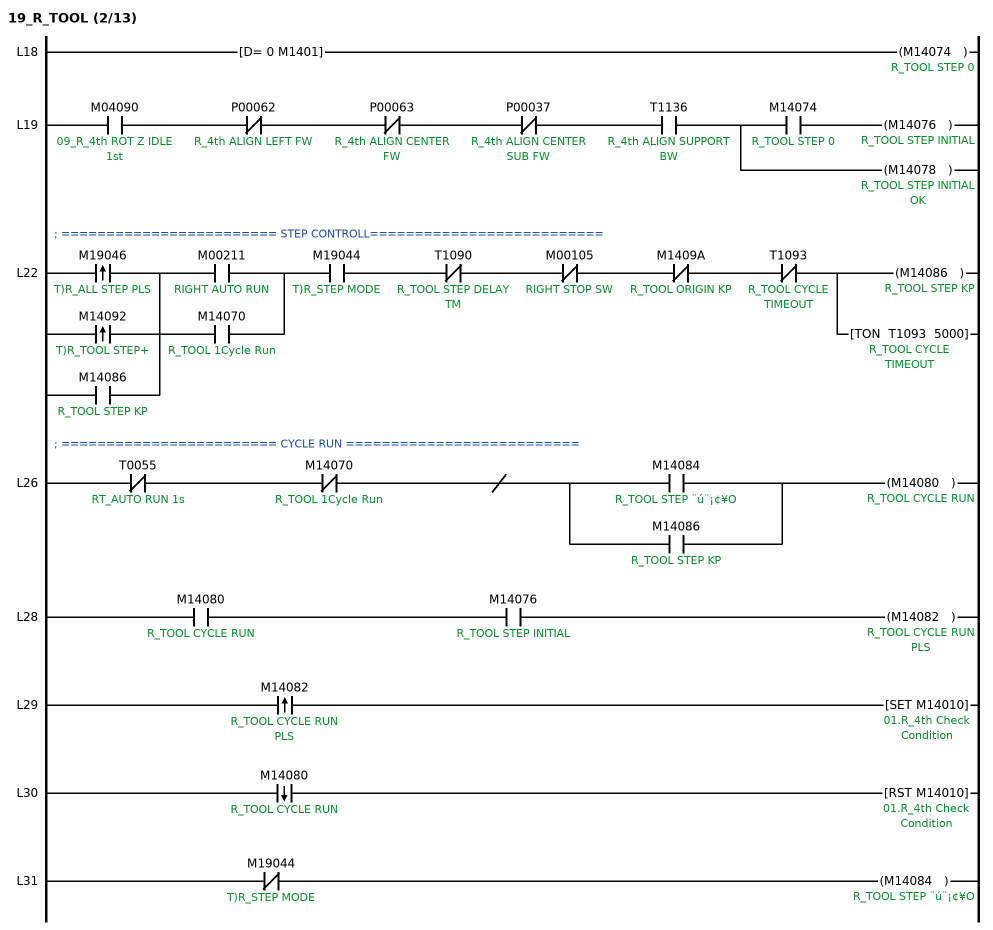
; L18
LOADD=    0 M1401
OUT       M14074	// R_TOOL STEP 0
; L19
LOAD      M04090	// 09_R_4th ROT Z IDLE 1st
AND NOT   P00062	// R_4th ALIGN LEFT FW
AND NOT   P00063	// R_4th ALIGN CENTER FW
AND NOT   P00037	// R_4th ALIGN CENTER SUB FW
AND       T1136	// R_4th ALIGN SUPPORT BW
MPUSH
AND       M14074	// R_TOOL STEP 0
OUT       M14076	// R_TOOL STEP INITIAL
MPOP
OUT       M14078	// R_TOOL STEP INITIAL OK
// ======================== STEP CONTROLL==========================
; L22
LOADP     M19046	// T)R_ALL STEP PLS
ORP       M14092	// T)R_TOOL STEP+
OR        M14086	// R_TOOL STEP KP
LOAD      M00211	// RIGHT AUTO RUN
OR        M14070	// R_TOOL 1Cycle Run
AND LOAD
AND       M19044	// T)R_STEP MODE
AND NOT   T1090	// R_TOOL STEP DELAY TM
AND NOT   M00105	// RIGHT STOP SW
AND NOT   M1409A	// R_TOOL ORIGIN KP
AND NOT   T1093	// R_TOOL CYCLE TIMEOUT
OUT       M14086	// R_TOOL STEP KP
TON       T1093 5000	// R_TOOL CYCLE TIMEOUT
// ======================== CYCLE RUN ==========================
; L26
LOAD NOT  T0055	// RT_AUTO RUN 1s
AND NOT   M14070	// R_TOOL 1Cycle Run
NOT
LOAD      M14084	// R_TOOL STEP ¨ú¨¡¢¥O
OR        M14086	// R_TOOL STEP KP
AND LOAD
OUT       M14080	// R_TOOL CYCLE RUN
; L28
LOAD      M14080	// R_TOOL CYCLE RUN
AND       M14076	// R_TOOL STEP INITIAL
OUT       M14082	// R_TOOL CYCLE RUN PLS
; L29
LOADP     M14082	// R_TOOL CYCLE RUN PLS
SET       M14010	// 01.R_4th Check Condition
; L30
LOADN     M14080	// R_TOOL CYCLE RUN
RST       M14010	// 01.R_4th Check Condition
; L31
LOAD NOT  M19044	// T)R_STEP MODE
OUT       M14084	// R_TOOL STEP ¨ú¨¡¢¥O

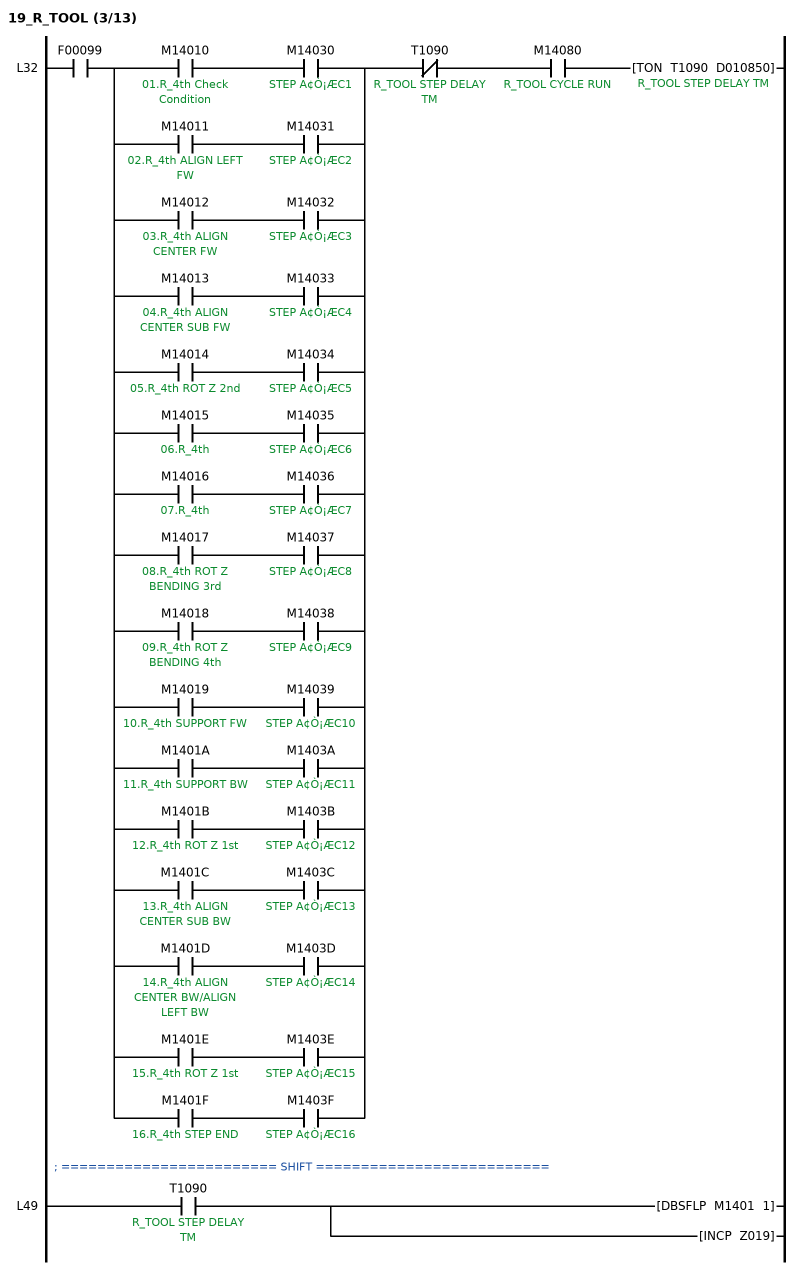
; L32
LOAD      F00099
LOAD      M14010	// 01.R_4th Check Condition
AND       M14030	// STEP A¢Ò¡ÆC1
LOAD      M14011	// 02.R_4th ALIGN LEFT FW
AND       M14031	// STEP A¢Ò¡ÆC2
OR LOAD
LOAD      M14012	// 03.R_4th ALIGN CENTER FW
AND       M14032	// STEP A¢Ò¡ÆC3
OR LOAD
LOAD      M14013	// 04.R_4th ALIGN CENTER SUB FW
AND       M14033	// STEP A¢Ò¡ÆC4
OR LOAD
LOAD      M14014	// 05.R_4th ROT Z 2nd
AND       M14034	// STEP A¢Ò¡ÆC5
OR LOAD
LOAD      M14015	// 06.R_4th
AND       M14035	// STEP A¢Ò¡ÆC6
OR LOAD
LOAD      M14016	// 07.R_4th 
AND       M14036	// STEP A¢Ò¡ÆC7
OR LOAD
LOAD      M14017	// 08.R_4th ROT Z BENDING 3rd
AND       M14037	// STEP A¢Ò¡ÆC8
OR LOAD
LOAD      M14018	// 09.R_4th ROT Z BENDING 4th
AND       M14038	// STEP A¢Ò¡ÆC9
OR LOAD
LOAD      M14019	// 10.R_4th SUPPORT FW
AND       M14039	// STEP A¢Ò¡ÆC10
OR LOAD
LOAD      M1401A	// 11.R_4th SUPPORT BW
AND       M1403A	// STEP A¢Ò¡ÆC11
OR LOAD
LOAD      M1401B	// 12.R_4th ROT Z 1st
AND       M1403B	// STEP A¢Ò¡ÆC12
OR LOAD
LOAD      M1401C	// 13.R_4th ALIGN CENTER SUB BW
AND       M1403C	// STEP A¢Ò¡ÆC13
OR LOAD
LOAD      M1401D	// 14.R_4th ALIGN CENTER BW/ALIGN LEFT BW
AND       M1403D	// STEP A¢Ò¡ÆC14
OR LOAD
LOAD      M1401E	// 15.R_4th ROT Z 1st
AND       M1403E	// STEP A¢Ò¡ÆC15
OR LOAD
LOAD      M1401F	// 16.R_4th STEP END
AND       M1403F	// STEP A¢Ò¡ÆC16
OR LOAD
AND LOAD
AND NOT   T1090	// R_TOOL STEP DELAY TM
AND       M14080	// R_TOOL CYCLE RUN
TON       T1090 D010850	// R_TOOL STEP DELAY TM
// ======================== SHIFT ==========================
; L49
LOAD      T1090	// R_TOOL STEP DELAY TM
DBSFLP    M1401 1
INCP      Z019

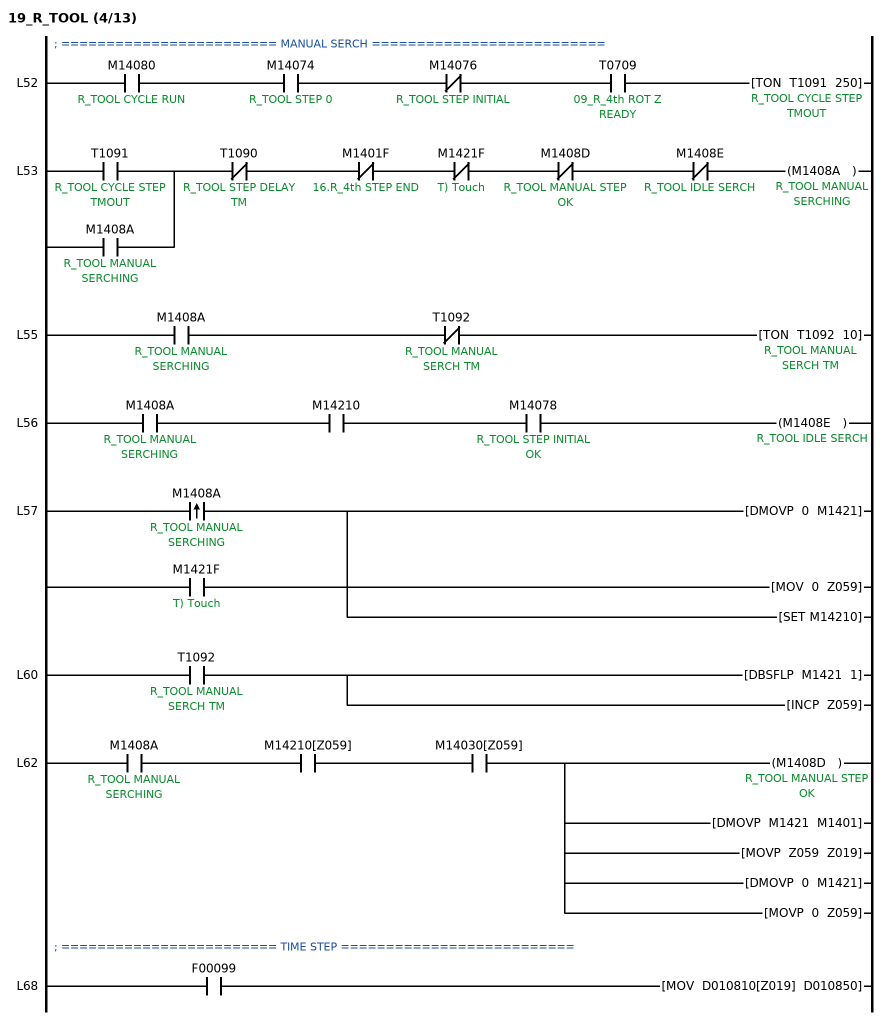
// ======================== MANUAL SERCH ==========================
; L52
LOAD      M14080	// R_TOOL CYCLE RUN
AND       M14074	// R_TOOL STEP 0
AND NOT   M14076	// R_TOOL STEP INITIAL
AND       T0709	// 09_R_4th ROT Z READY
TON       T1091 250	// R_TOOL CYCLE STEP TMOUT
; L53
LOAD      T1091	// R_TOOL CYCLE STEP TMOUT
OR        M1408A	// R_TOOL MANUAL SERCHING
AND NOT   T1090	// R_TOOL STEP DELAY TM
AND NOT   M1401F	// 16.R_4th STEP END
AND NOT   M1421F	// T) Touch
AND NOT   M1408D	// R_TOOL MANUAL STEP OK
AND NOT   M1408E	// R_TOOL IDLE SERCH
OUT       M1408A	// R_TOOL MANUAL SERCHING
; L55
LOAD      M1408A	// R_TOOL MANUAL SERCHING
AND NOT   T1092	// R_TOOL MANUAL SERCH TM
TON       T1092 10	// R_TOOL MANUAL SERCH TM
; L56
LOAD      M1408A	// R_TOOL MANUAL SERCHING
AND       M14210
AND       M14078	// R_TOOL STEP INITIAL OK
OUT       M1408E	// R_TOOL IDLE SERCH
; L57
LOADP     M1408A	// R_TOOL MANUAL SERCHING
OR        M1421F	// T) Touch
DMOVP     0 M1421
MOV       0 Z059
SET       M14210
; L60
LOAD      T1092	// R_TOOL MANUAL SERCH TM
DBSFLP    M1421 1
INCP      Z059
; L62
LOAD      M1408A	// R_TOOL MANUAL SERCHING
AND       M14210[Z059]
AND       M14030[Z059]
OUT       M1408D	// R_TOOL MANUAL STEP OK
DMOVP     M1421 M1401
MOVP      Z059 Z019
DMOVP     0 M1421
MOVP      0 Z059
// ======================== TIME STEP ==========================
; L68
LOAD      F00099
MOV       D010810[Z019] D010850

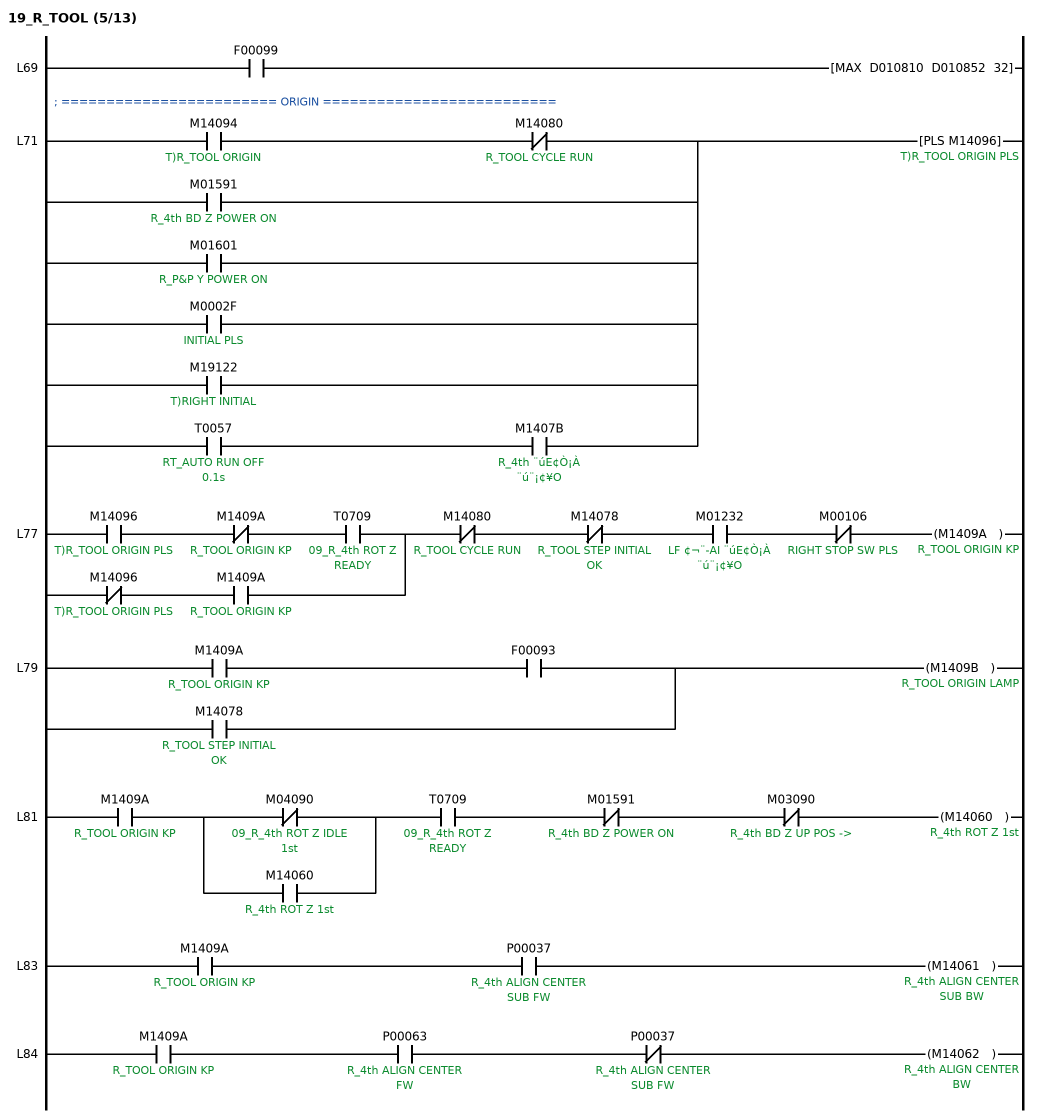
; L69
LOAD      F00099
MAX       D010810 D010852 32
// ======================== ORIGIN ==========================
; L71
LOAD      M14094	// T)R_TOOL ORIGIN
AND NOT   M14080	// R_TOOL CYCLE RUN
OR        M01591	// R_4th BD Z POWER ON
OR        M01601	// R_P&P Y POWER ON
OR        M0002F	// INITIAL PLS
OR        M19122	// T)RIGHT INITIAL
LOAD      T0057	// RT_AUTO RUN OFF 0.1s
AND       M1407B	// R_4th ¨úE¢Ò¡À ¨ú¨¡¢¥O
OR LOAD
OUTP      M14096	// T)R_TOOL ORIGIN PLS
; L77
LOAD      M14096	// T)R_TOOL ORIGIN PLS
AND NOT   M1409A	// R_TOOL ORIGIN KP
AND       T0709	// 09_R_4th ROT Z READY
LOAD NOT  M14096	// T)R_TOOL ORIGIN PLS
AND       M1409A	// R_TOOL ORIGIN KP
OR LOAD
AND NOT   M14080	// R_TOOL CYCLE RUN
AND NOT   M14078	// R_TOOL STEP INITIAL OK
AND       M01232	// LF ¢¬¨­AI ¨úE¢Ò¡À ¨ú¨¡¢¥O
AND NOT   M00106	// RIGHT STOP SW PLS
OUT       M1409A	// R_TOOL ORIGIN KP
; L79
LOAD      M1409A	// R_TOOL ORIGIN KP
AND       F00093
OR        M14078	// R_TOOL STEP INITIAL OK
OUT       M1409B	// R_TOOL ORIGIN LAMP
; L81
LOAD      M1409A	// R_TOOL ORIGIN KP
LOAD NOT  M04090	// 09_R_4th ROT Z IDLE 1st
OR        M14060	// R_4th ROT Z 1st
AND LOAD
AND       T0709	// 09_R_4th ROT Z READY
AND NOT   M01591	// R_4th BD Z POWER ON
AND NOT   M03090	// R_4th BD Z UP POS ->
OUT       M14060	// R_4th ROT Z 1st
; L83
LOAD      M1409A	// R_TOOL ORIGIN KP
AND       P00037	// R_4th ALIGN CENTER SUB FW
OUT       M14061	// R_4th ALIGN CENTER SUB BW
; L84
LOAD      M1409A	// R_TOOL ORIGIN KP
AND       P00063	// R_4th ALIGN CENTER FW
AND NOT   P00037	// R_4th ALIGN CENTER SUB FW
OUT       M14062	// R_4th ALIGN CENTER BW

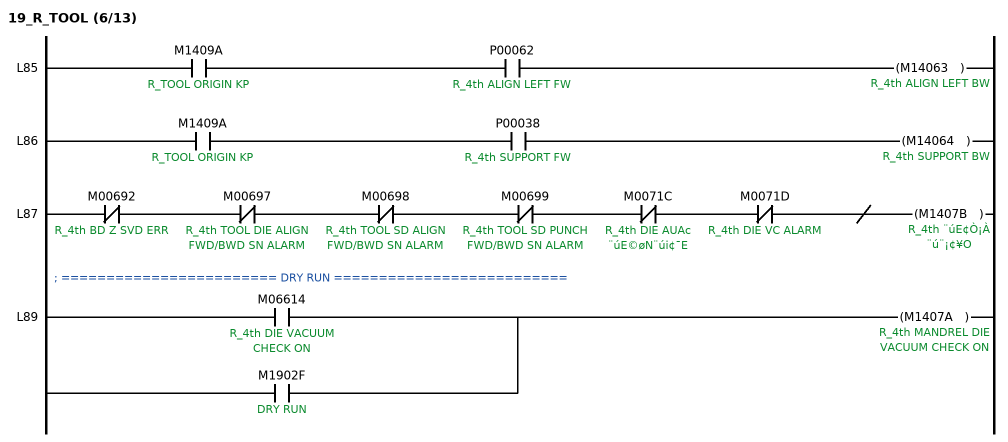
; L85
LOAD      M1409A	// R_TOOL ORIGIN KP
AND       P00062	// R_4th ALIGN LEFT FW
OUT       M14063	// R_4th ALIGN LEFT BW
; L86
LOAD      M1409A	// R_TOOL ORIGIN KP
AND       P00038	// R_4th SUPPORT FW
OUT       M14064	// R_4th SUPPORT BW
; L87
LOAD NOT  M00692	// R_4th BD Z SVD ERR
AND NOT   M00697	// R_4th TOOL DIE ALIGN FWD/BWD SN ALARM
AND NOT   M00698	// R_4th TOOL SD ALIGN FWD/BWD SN ALARM
AND NOT   M00699	// R_4th TOOL SD PUNCH FWD/BWD SN ALARM
AND NOT   M0071C	// R_4th DIE AUAc ¨úE©øN¨úi¢¯E
AND NOT   M0071D	// R_4th DIE VC ALARM
NOT
OUT       M1407B	// R_4th ¨úE¢Ò¡À ¨ú¨¡¢¥O
// ======================== DRY RUN ==========================
; L89
LOAD      M06614	// R_4th DIE VACUUM CHECK ON
OR        M1902F	// DRY RUN
OUT       M1407A	// R_4th MANDREL DIE VACUUM CHECK ON

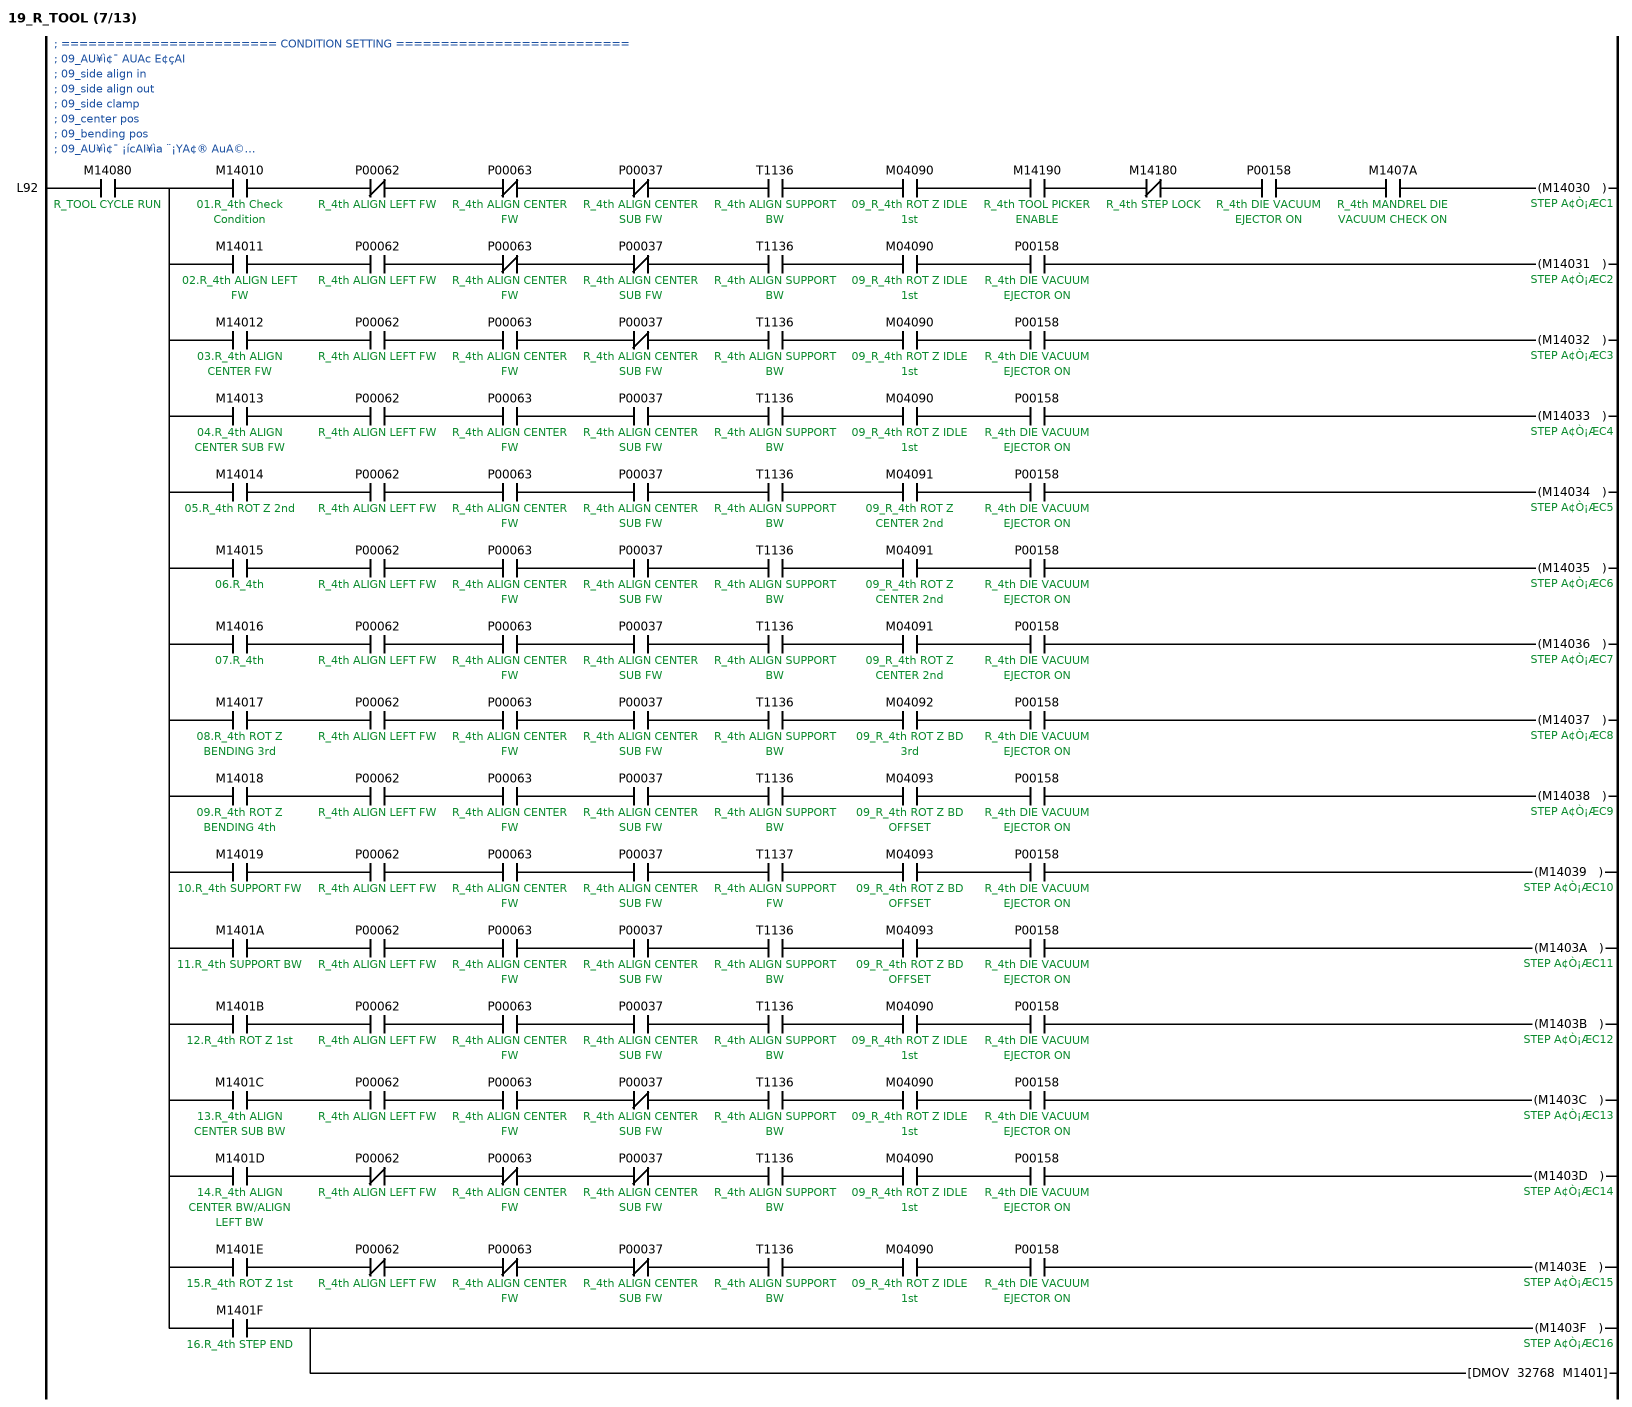
// ======================== CONDITION SETTING ==========================
; L92
LOAD      M14080	// R_TOOL CYCLE RUN
MPUSH
AND       M14010	// 01.R_4th Check Condition
AND NOT   P00062	// R_4th ALIGN LEFT FW
AND NOT   P00063	// R_4th ALIGN CENTER FW
AND NOT   P00037	// R_4th ALIGN CENTER SUB FW
AND       T1136	// R_4th ALIGN SUPPORT BW
AND       M04090	// 09_R_4th ROT Z IDLE 1st
AND       M14190	// R_4th TOOL PICKER ENABLE
AND NOT   M14180	// R_4th STEP LOCK
AND       P00158	// R_4th DIE VACUUM EJECTOR ON
AND       M1407A	// R_4th MANDREL DIE VACUUM CHECK ON
OUT       M14030	// STEP A¢Ò¡ÆC1
MLOAD
AND       M14011	// 02.R_4th ALIGN LEFT FW
AND       P00062	// R_4th ALIGN LEFT FW
AND NOT   P00063	// R_4th ALIGN CENTER FW
AND NOT   P00037	// R_4th ALIGN CENTER SUB FW
AND       T1136	// R_4th ALIGN SUPPORT BW
AND       M04090	// 09_R_4th ROT Z IDLE 1st
AND       P00158	// R_4th DIE VACUUM EJECTOR ON
OUT       M14031	// STEP A¢Ò¡ÆC2
MLOAD
AND       M14012	// 03.R_4th ALIGN CENTER FW
AND       P00062	// R_4th ALIGN LEFT FW
AND       P00063	// R_4th ALIGN CENTER FW
AND NOT   P00037	// R_4th ALIGN CENTER SUB FW
AND       T1136	// R_4th ALIGN SUPPORT BW
AND       M04090	// 09_R_4th ROT Z IDLE 1st
AND       P00158	// R_4th DIE VACUUM EJECTOR ON
OUT       M14032	// STEP A¢Ò¡ÆC3
MLOAD
AND       M14013	// 04.R_4th ALIGN CENTER SUB FW
AND       P00062	// R_4th ALIGN LEFT FW
AND       P00063	// R_4th ALIGN CENTER FW
AND       P00037	// R_4th ALIGN CENTER SUB FW
AND       T1136	// R_4th ALIGN SUPPORT BW
AND       M04090	// 09_R_4th ROT Z IDLE 1st
AND       P00158	// R_4th DIE VACUUM EJECTOR ON
OUT       M14033	// STEP A¢Ò¡ÆC4
MLOAD
AND       M14014	// 05.R_4th ROT Z 2nd
AND       P00062	// R_4th ALIGN LEFT FW
AND       P00063	// R_4th ALIGN CENTER FW
AND       P00037	// R_4th ALIGN CENTER SUB FW
AND       T1136	// R_4th ALIGN SUPPORT BW
AND       M04091	// 09_R_4th ROT Z CENTER 2nd
AND       P00158	// R_4th DIE VACUUM EJECTOR ON
OUT       M14034	// STEP A¢Ò¡ÆC5
MLOAD
AND       M14015	// 06.R_4th
AND       P00062	// R_4th ALIGN LEFT FW
AND       P00063	// R_4th ALIGN CENTER FW
AND       P00037	// R_4th ALIGN CENTER SUB FW
AND       T1136	// R_4th ALIGN SUPPORT BW
AND       M04091	// 09_R_4th ROT Z CENTER 2nd
AND       P00158	// R_4th DIE VACUUM EJECTOR ON
OUT       M14035	// STEP A¢Ò¡ÆC6
MLOAD
AND       M14016	// 07.R_4th 
AND       P00062	// R_4th ALIGN LEFT FW
AND       P00063	// R_4th ALIGN CENTER FW
AND       P00037	// R_4th ALIGN CENTER SUB FW
AND       T1136	// R_4th ALIGN SUPPORT BW
AND       M04091	// 09_R_4th ROT Z CENTER 2nd
AND       P00158	// R_4th DIE VACUUM EJECTOR ON
OUT       M14036	// STEP A¢Ò¡ÆC7
MLOAD
AND       M14017	// 08.R_4th ROT Z BENDING 3rd
AND       P00062	// R_4th ALIGN LEFT FW
AND       P00063	// R_4th ALIGN CENTER FW
AND       P00037	// R_4th ALIGN CENTER SUB FW
AND       T1136	// R_4th ALIGN SUPPORT BW
AND       M04092	// 09_R_4th ROT Z BD 3rd
AND       P00158	// R_4th DIE VACUUM EJECTOR ON
OUT       M14037	// STEP A¢Ò¡ÆC8
MLOAD
AND       M14018	// 09.R_4th ROT Z BENDING 4th
AND       P00062	// R_4th ALIGN LEFT FW
AND       P00063	// R_4th ALIGN CENTER FW
AND       P00037	// R_4th ALIGN CENTER SUB FW
AND       T1136	// R_4th ALIGN SUPPORT BW
AND       M04093	// 09_R_4th ROT Z BD OFFSET
AND       P00158	// R_4th DIE VACUUM EJECTOR ON
OUT       M14038	// STEP A¢Ò¡ÆC9
MLOAD
AND       M14019	// 10.R_4th SUPPORT FW
AND       P00062	// R_4th ALIGN LEFT FW
AND       P00063	// R_4th ALIGN CENTER FW
AND       P00037	// R_4th ALIGN CENTER SUB FW
AND       T1137	// R_4th ALIGN SUPPORT FW
AND       M04093	// 09_R_4th ROT Z BD OFFSET
AND       P00158	// R_4th DIE VACUUM EJECTOR ON
OUT       M14039	// STEP A¢Ò¡ÆC10
MLOAD
AND       M1401A	// 11.R_4th SUPPORT BW
AND       P00062	// R_4th ALIGN LEFT FW
AND       P00063	// R_4th ALIGN CENTER FW
AND       P00037	// R_4th ALIGN CENTER SUB FW
AND       T1136	// R_4th ALIGN SUPPORT BW
AND       M04093	// 09_R_4th ROT Z BD OFFSET
AND       P00158	// R_4th DIE VACUUM EJECTOR ON
OUT       M1403A	// STEP A¢Ò¡ÆC11
MLOAD
AND       M1401B	// 12.R_4th ROT Z 1st
AND       P00062	// R_4th ALIGN LEFT FW
AND       P00063	// R_4th ALIGN CENTER FW
AND       P00037	// R_4th ALIGN CENTER SUB FW
AND       T1136	// R_4th ALIGN SUPPORT BW
AND       M04090	// 09_R_4th ROT Z IDLE 1st
AND       P00158	// R_4th DIE VACUUM EJECTOR ON
OUT       M1403B	// STEP A¢Ò¡ÆC12
MLOAD
AND       M1401C	// 13.R_4th ALIGN CENTER SUB BW
AND       P00062	// R_4th ALIGN LEFT FW
AND       P00063	// R_4th ALIGN CENTER FW
AND NOT   P00037	// R_4th ALIGN CENTER SUB FW
AND       T1136	// R_4th ALIGN SUPPORT BW
AND       M04090	// 09_R_4th ROT Z IDLE 1st
AND       P00158	// R_4th DIE VACUUM EJECTOR ON
OUT       M1403C	// STEP A¢Ò¡ÆC13
MLOAD
AND       M1401D	// 14.R_4th ALIGN CENTER BW/ALIGN LEFT BW
AND NOT   P00062	// R_4th ALIGN LEFT FW
AND NOT   P00063	// R_4th ALIGN CENTER FW
AND NOT   P00037	// R_4th ALIGN CENTER SUB FW
AND       T1136	// R_4th ALIGN SUPPORT BW
AND       M04090	// 09_R_4th ROT Z IDLE 1st
AND       P00158	// R_4th DIE VACUUM EJECTOR ON
OUT       M1403D	// STEP A¢Ò¡ÆC14
MLOAD
AND       M1401E	// 15.R_4th ROT Z 1st
AND NOT   P00062	// R_4th ALIGN LEFT FW
AND NOT   P00063	// R_4th ALIGN CENTER FW
AND NOT   P00037	// R_4th ALIGN CENTER SUB FW
AND       T1136	// R_4th ALIGN SUPPORT BW
AND       M04090	// 09_R_4th ROT Z IDLE 1st
AND       P00158	// R_4th DIE VACUUM EJECTOR ON
OUT       M1403E	// STEP A¢Ò¡ÆC15
MPOP
AND       M1401F	// 16.R_4th STEP END
OUT       M1403F	// STEP A¢Ò¡ÆC16
DMOV      32768 M1401
// output comment: 09_AU¥ì¢¯ AUAc E¢çAI
// output comment: 09_side align in
// output comment: 09_side align out
// output comment: 09_side clamp
// output comment: 09_center pos
// output comment: 09_bending pos
// output comment: 09_AU¥ì¢¯ ¡ícAI¥ìa ¨¡YA¢® AuA©ª
// output comment: 09_AU¥ì¢¯ ¡ícAI¥ìa ¨¡YA¢® EAA©ª(X1652) 09_AU¥ì¢¯ Z ¡ío¨öA A¡×A¢® -> (X1666)
// output comment: 09_AU¥ì¢¯ ¡ícAI¥ìa ¨¡YA¢® EAA©ª(X1666) 09_AU¥ì¢¯ Z ¡ío¨öA A¡×A¢® -> (X1652)

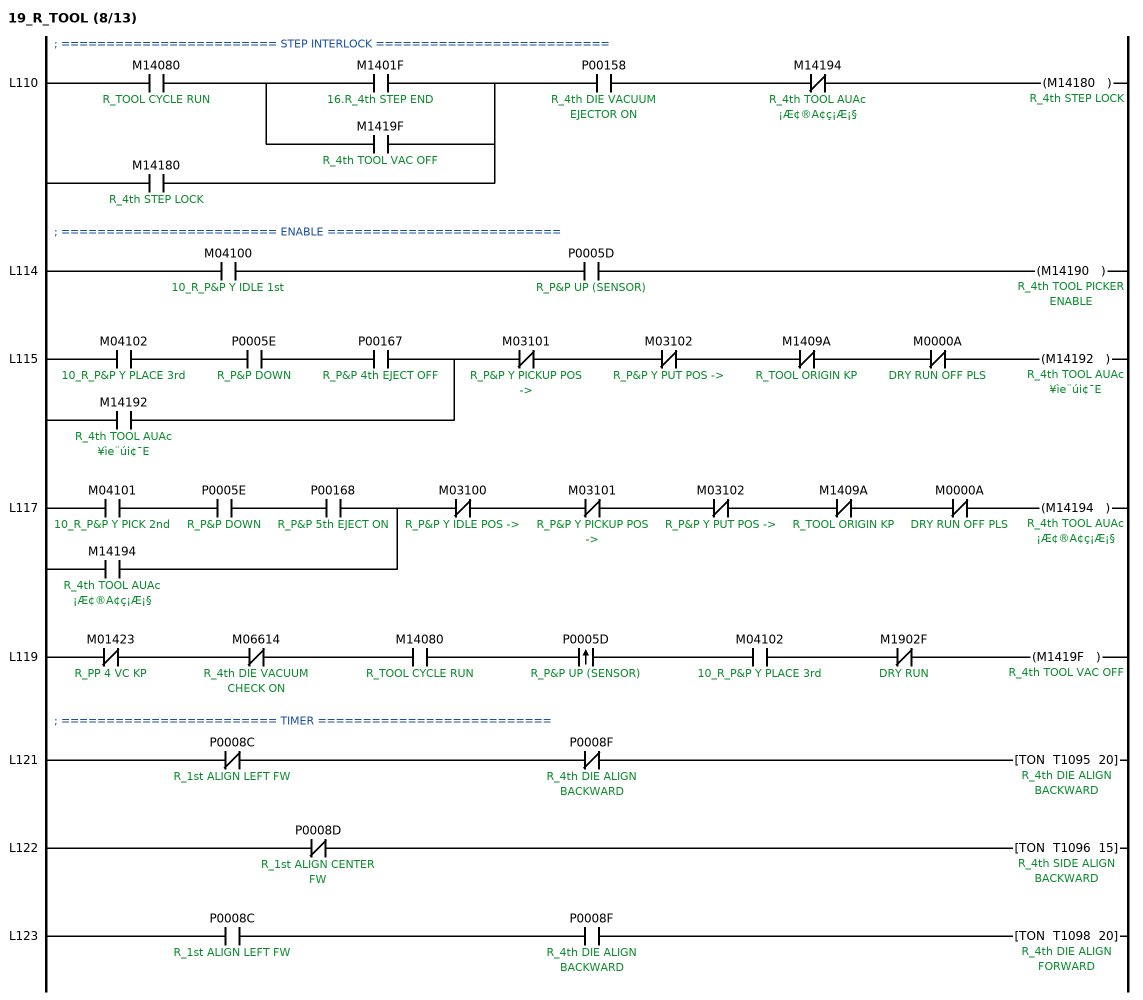
// ======================== STEP INTERLOCK ==========================
; L110
LOAD      M14080	// R_TOOL CYCLE RUN
LOAD      M1401F	// 16.R_4th STEP END
OR        M1419F	// R_4th TOOL VAC OFF
AND LOAD
OR        M14180	// R_4th STEP LOCK
AND       P00158	// R_4th DIE VACUUM EJECTOR ON
AND NOT   M14194	// R_4th TOOL AUAc ¡Æ¢®A¢ç¡Æ¡§
OUT       M14180	// R_4th STEP LOCK
// ======================== ENABLE ==========================
; L114
LOAD      M04100	// 10_R_P&P Y IDLE 1st
AND       P0005D	// R_P&P UP (SENSOR)
OUT       M14190	// R_4th TOOL PICKER ENABLE
; L115
LOAD      M04102	// 10_R_P&P Y PLACE 3rd
AND       P0005E	// R_P&P DOWN
AND       P00167	// R_P&P 4th EJECT OFF
OR        M14192	// R_4th TOOL AUAc ¥ìe¨úi¢¯E
AND NOT   M03101	// R_P&P Y PICKUP POS ->
AND NOT   M03102	// R_P&P Y PUT POS ->
AND NOT   M1409A	// R_TOOL ORIGIN KP
AND NOT   M0000A	// DRY RUN OFF PLS
OUT       M14192	// R_4th TOOL AUAc ¥ìe¨úi¢¯E
; L117
LOAD      M04101	// 10_R_P&P Y PICK 2nd
AND       P0005E	// R_P&P DOWN
AND       P00168	// R_P&P 5th EJECT ON
OR        M14194	// R_4th TOOL AUAc ¡Æ¢®A¢ç¡Æ¡§
AND NOT   M03100	// R_P&P Y IDLE POS ->
AND NOT   M03101	// R_P&P Y PICKUP POS ->
AND NOT   M03102	// R_P&P Y PUT POS ->
AND NOT   M1409A	// R_TOOL ORIGIN KP
AND NOT   M0000A	// DRY RUN OFF PLS
OUT       M14194	// R_4th TOOL AUAc ¡Æ¢®A¢ç¡Æ¡§
; L119
LOAD NOT  M01423	// R_PP 4 VC KP
AND NOT   M06614	// R_4th DIE VACUUM CHECK ON
AND       M14080	// R_TOOL CYCLE RUN
ANDP      P0005D	// R_P&P UP (SENSOR)
AND       M04102	// 10_R_P&P Y PLACE 3rd
AND NOT   M1902F	// DRY RUN
OUT       M1419F	// R_4th TOOL VAC OFF
// ======================== TIMER ==========================
; L121
LOAD NOT  P0008C	// R_1st ALIGN LEFT FW
AND NOT   P0008F	// R_4th DIE ALIGN BACKWARD
TON       T1095 20	// R_4th DIE ALIGN BACKWARD
; L122
LOAD NOT  P0008D	// R_1st ALIGN CENTER FW
TON       T1096 15	// R_4th SIDE ALIGN BACKWARD
; L123
LOAD      P0008C	// R_1st ALIGN LEFT FW
AND       P0008F	// R_4th DIE ALIGN BACKWARD
TON       T1098 20	// R_4th DIE ALIGN FORWARD

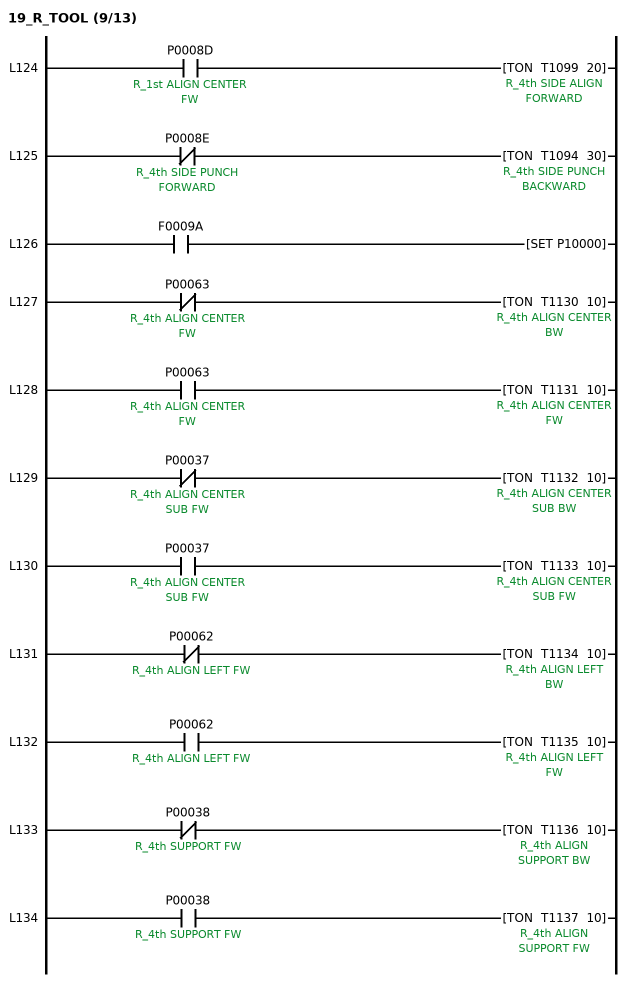
; L124
LOAD      P0008D	// R_1st ALIGN CENTER FW
TON       T1099 20	// R_4th SIDE ALIGN FORWARD
; L125
LOAD NOT  P0008E	// R_4th SIDE PUNCH FORWARD
TON       T1094 30	// R_4th SIDE PUNCH BACKWARD
; L126
LOAD      F0009A
SET       P10000
; L127
LOAD NOT  P00063	// R_4th ALIGN CENTER FW
TON       T1130 10	// R_4th ALIGN CENTER BW
; L128
LOAD      P00063	// R_4th ALIGN CENTER FW
TON       T1131 10	// R_4th ALIGN CENTER FW
; L129
LOAD NOT  P00037	// R_4th ALIGN CENTER SUB FW
TON       T1132 10	// R_4th ALIGN CENTER SUB BW
; L130
LOAD      P00037	// R_4th ALIGN CENTER SUB FW
TON       T1133 10	// R_4th ALIGN CENTER SUB FW
; L131
LOAD NOT  P00062	// R_4th ALIGN LEFT FW
TON       T1134 10	// R_4th ALIGN LEFT BW
; L132
LOAD      P00062	// R_4th ALIGN LEFT FW
TON       T1135 10	// R_4th ALIGN LEFT FW
; L133
LOAD NOT  P00038	// R_4th SUPPORT FW
TON       T1136 10	// R_4th ALIGN SUPPORT BW
; L134
LOAD      P00038	// R_4th SUPPORT FW
TON       T1137 10	// R_4th ALIGN SUPPORT FW

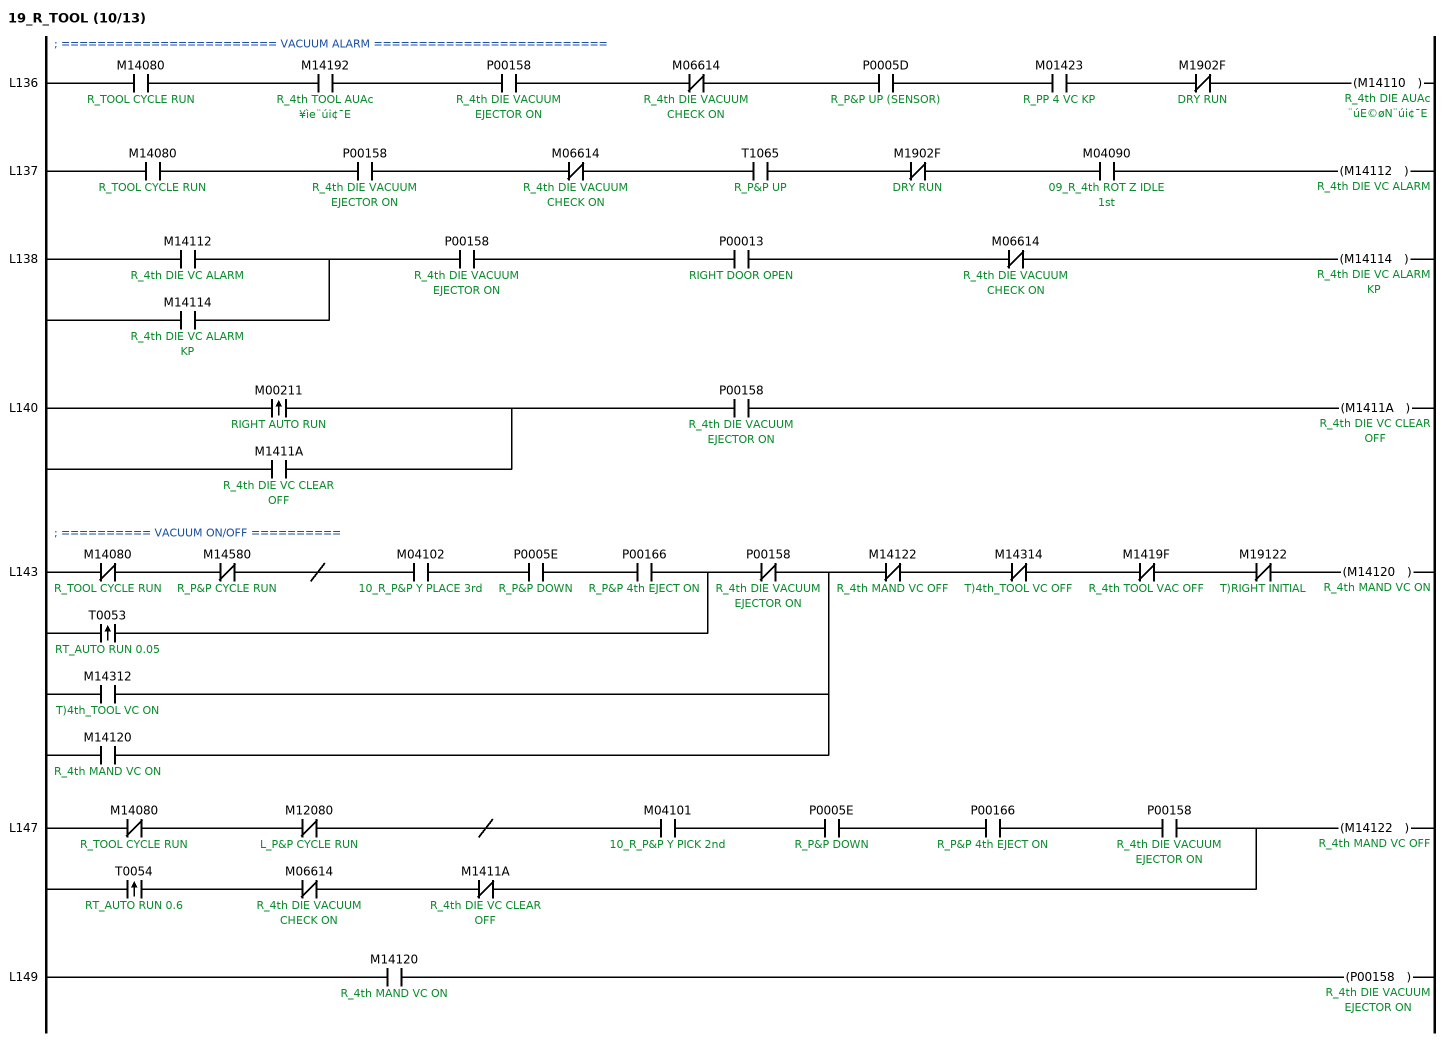
// ======================== VACUUM ALARM ==========================
; L136
LOAD      M14080	// R_TOOL CYCLE RUN
AND       M14192	// R_4th TOOL AUAc ¥ìe¨úi¢¯E
AND       P00158	// R_4th DIE VACUUM EJECTOR ON
AND NOT   M06614	// R_4th DIE VACUUM CHECK ON
AND       P0005D	// R_P&P UP (SENSOR)
AND       M01423	// R_PP 4 VC KP
AND NOT   M1902F	// DRY RUN
OUT       M14110	// R_4th DIE AUAc ¨úE©øN¨úi¢¯E
; L137
LOAD      M14080	// R_TOOL CYCLE RUN
AND       P00158	// R_4th DIE VACUUM EJECTOR ON
AND NOT   M06614	// R_4th DIE VACUUM CHECK ON
AND       T1065	// R_P&P UP
AND NOT   M1902F	// DRY RUN
AND       M04090	// 09_R_4th ROT Z IDLE 1st
OUT       M14112	// R_4th DIE VC ALARM
; L138
LOAD      M14112	// R_4th DIE VC ALARM
OR        M14114	// R_4th DIE VC ALARM KP
AND       P00158	// R_4th DIE VACUUM EJECTOR ON
AND       P00013	// RIGHT DOOR OPEN
AND NOT   M06614	// R_4th DIE VACUUM CHECK ON
OUT       M14114	// R_4th DIE VC ALARM KP
; L140
LOADP     M00211	// RIGHT AUTO RUN
OR        M1411A	// R_4th DIE VC CLEAR OFF
AND       P00158	// R_4th DIE VACUUM EJECTOR ON
OUT       M1411A	// R_4th DIE VC CLEAR OFF
// ========== VACUUM ON/OFF ==========
; L143
LOAD NOT  M14080	// R_TOOL CYCLE RUN
AND NOT   M14580	// R_P&P CYCLE RUN
NOT
AND       M04102	// 10_R_P&P Y PLACE 3rd
AND       P0005E	// R_P&P DOWN
AND       P00166	// R_P&P 4th EJECT ON
ORP       T0053	// RT_AUTO RUN 0.05
AND NOT   P00158	// R_4th DIE VACUUM EJECTOR ON
OR        M14312	// T)4th_TOOL VC ON
OR        M14120	// R_4th MAND VC ON
AND NOT   M14122	// R_4th MAND VC OFF
AND NOT   M14314	// T)4th_TOOL VC OFF
AND NOT   M1419F	// R_4th TOOL VAC OFF
AND NOT   M19122	// T)RIGHT INITIAL
OUT       M14120	// R_4th MAND VC ON
; L147
LOAD NOT  M14080	// R_TOOL CYCLE RUN
AND NOT   M12080	// L_P&P CYCLE RUN
NOT
AND       M04101	// 10_R_P&P Y PICK 2nd
AND       P0005E	// R_P&P DOWN
AND       P00166	// R_P&P 4th EJECT ON
AND       P00158	// R_4th DIE VACUUM EJECTOR ON
LOADP     T0054	// RT_AUTO RUN 0.6
AND NOT   M06614	// R_4th DIE VACUUM CHECK ON
AND NOT   M1411A	// R_4th DIE VC CLEAR OFF
OR LOAD
OUT       M14122	// R_4th MAND VC OFF
; L149
LOAD      M14120	// R_4th MAND VC ON
OUT       P00158	// R_4th DIE VACUUM EJECTOR ON

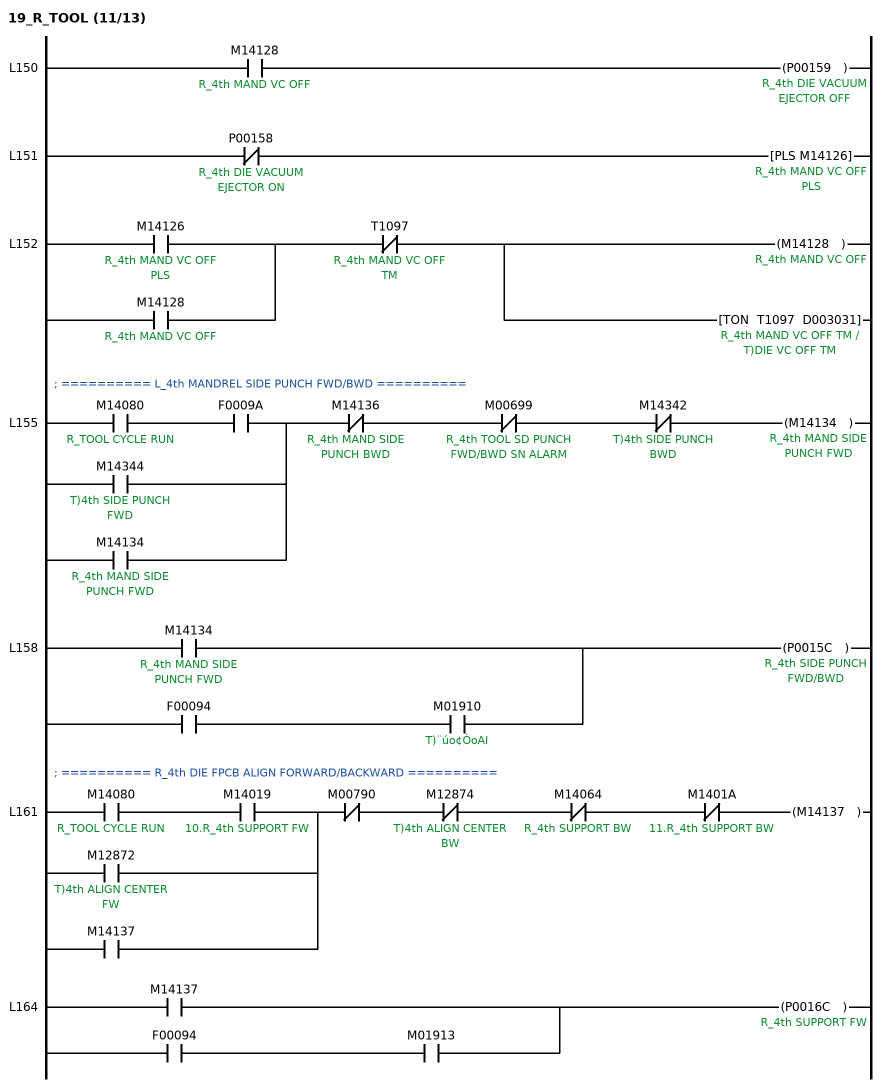
; L150
LOAD      M14128	// R_4th MAND VC OFF
OUT       P00159	// R_4th DIE VACUUM EJECTOR OFF
; L151
LOAD NOT  P00158	// R_4th DIE VACUUM EJECTOR ON
OUTP      M14126	// R_4th MAND VC OFF PLS
; L152
LOAD      M14126	// R_4th MAND VC OFF PLS
OR        M14128	// R_4th MAND VC OFF
AND NOT   T1097	// R_4th MAND VC OFF TM
OUT       M14128	// R_4th MAND VC OFF
TON       T1097 D003031	// R_4th MAND VC OFF TM / T)DIE VC OFF TM
// ========== L_4th MANDREL SIDE PUNCH FWD/BWD ==========
; L155
LOAD      M14080	// R_TOOL CYCLE RUN
AND       F0009A
OR        M14344	// T)4th SIDE PUNCH FWD
OR        M14134	// R_4th MAND SIDE PUNCH FWD
AND NOT   M14136	// R_4th MAND SIDE PUNCH BWD
AND NOT   M00699	// R_4th TOOL SD PUNCH FWD/BWD SN ALARM
AND NOT   M14342	// T)4th SIDE PUNCH BWD
OUT       M14134	// R_4th MAND SIDE PUNCH FWD
; L158
LOAD      M14134	// R_4th MAND SIDE PUNCH FWD
LOAD      F00094
AND       M01910	// T)¨úo¢ÒoAI
OR LOAD
OUT       P0015C	// R_4th SIDE PUNCH FWD/BWD
// ========== R_4th DIE FPCB ALIGN FORWARD/BACKWARD ==========
; L161
LOAD      M14080	// R_TOOL CYCLE RUN
AND       M14019	// 10.R_4th SUPPORT FW
OR        M12872	// T)4th ALIGN CENTER FW
OR        M14137
AND NOT   M00790
AND NOT   M12874	// T)4th ALIGN CENTER BW
AND NOT   M14064	// R_4th SUPPORT BW
AND NOT   M1401A	// 11.R_4th SUPPORT BW
OUT       M14137
; L164
LOAD      M14137
LOAD      F00094
AND       M01913
OR LOAD
OUT       P0016C	// R_4th SUPPORT FW

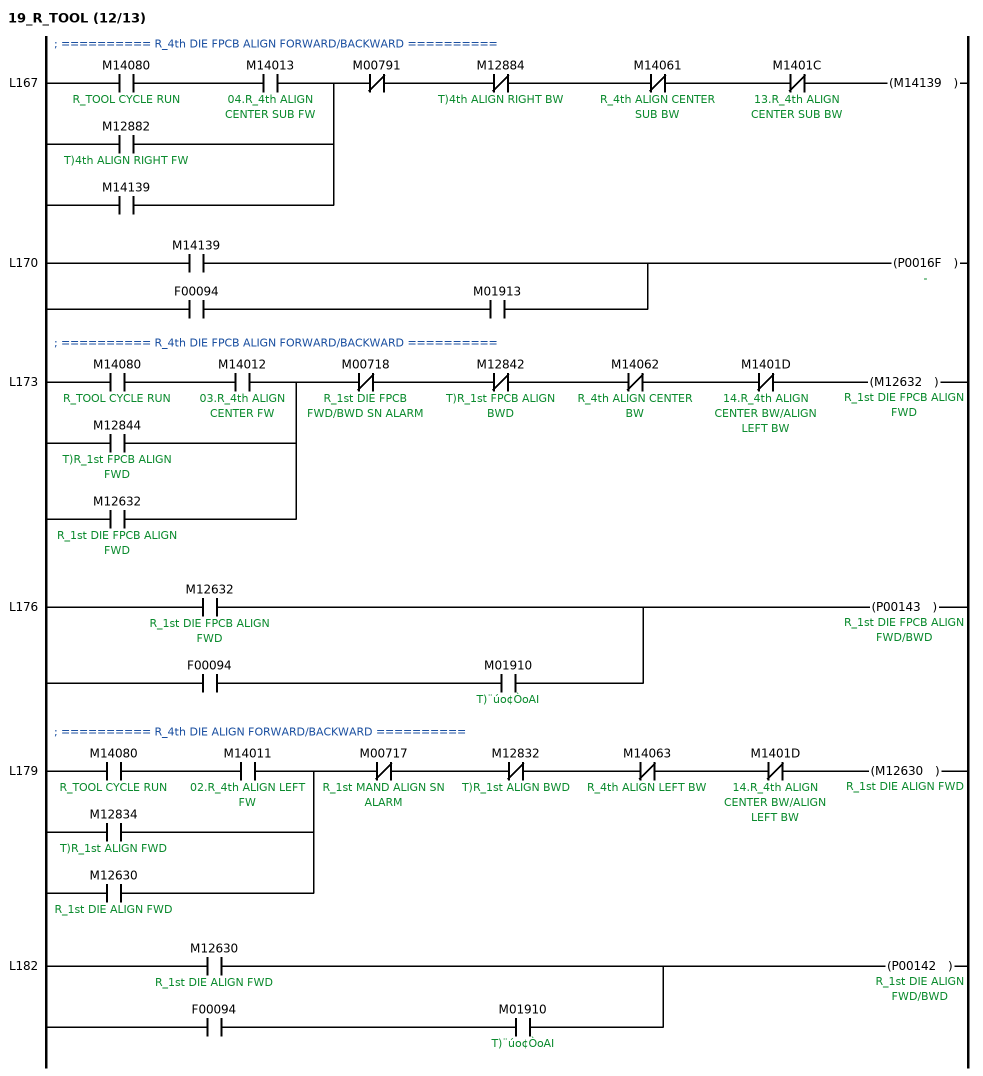
// ========== R_4th DIE FPCB ALIGN FORWARD/BACKWARD ==========
; L167
LOAD      M14080	// R_TOOL CYCLE RUN
AND       M14013	// 04.R_4th ALIGN CENTER SUB FW
OR        M12882	// T)4th ALIGN RIGHT FW
OR        M14139
AND NOT   M00791
AND NOT   M12884	// T)4th ALIGN RIGHT BW
AND NOT   M14061	// R_4th ALIGN CENTER SUB BW
AND NOT   M1401C	// 13.R_4th ALIGN CENTER SUB BW
OUT       M14139
; L170
LOAD      M14139
LOAD      F00094
AND       M01913
OR LOAD
OUT       P0016F	// -
// ========== R_4th DIE FPCB ALIGN FORWARD/BACKWARD ==========
; L173
LOAD      M14080	// R_TOOL CYCLE RUN
AND       M14012	// 03.R_4th ALIGN CENTER FW
OR        M12844	// T)R_1st FPCB ALIGN FWD
OR        M12632	// R_1st DIE FPCB ALIGN FWD
AND NOT   M00718	// R_1st DIE FPCB FWD/BWD SN ALARM
AND NOT   M12842	// T)R_1st FPCB ALIGN BWD
AND NOT   M14062	// R_4th ALIGN CENTER BW
AND NOT   M1401D	// 14.R_4th ALIGN CENTER BW/ALIGN LEFT BW
OUT       M12632	// R_1st DIE FPCB ALIGN FWD
; L176
LOAD      M12632	// R_1st DIE FPCB ALIGN FWD
LOAD      F00094
AND       M01910	// T)¨úo¢ÒoAI
OR LOAD
OUT       P00143	// R_1st DIE FPCB ALIGN FWD/BWD
// ========== R_4th DIE ALIGN FORWARD/BACKWARD ==========
; L179
LOAD      M14080	// R_TOOL CYCLE RUN
AND       M14011	// 02.R_4th ALIGN LEFT FW
OR        M12834	// T)R_1st ALIGN FWD
OR        M12630	// R_1st DIE ALIGN FWD
AND NOT   M00717	// R_1st MAND ALIGN SN ALARM
AND NOT   M12832	// T)R_1st ALIGN BWD
AND NOT   M14063	// R_4th ALIGN LEFT BW
AND NOT   M1401D	// 14.R_4th ALIGN CENTER BW/ALIGN LEFT BW
OUT       M12630	// R_1st DIE ALIGN FWD
; L182
LOAD      M12630	// R_1st DIE ALIGN FWD
LOAD      F00094
AND       M01910	// T)¨úo¢ÒoAI
OR LOAD
OUT       P00142	// R_1st DIE ALIGN FWD/BWD

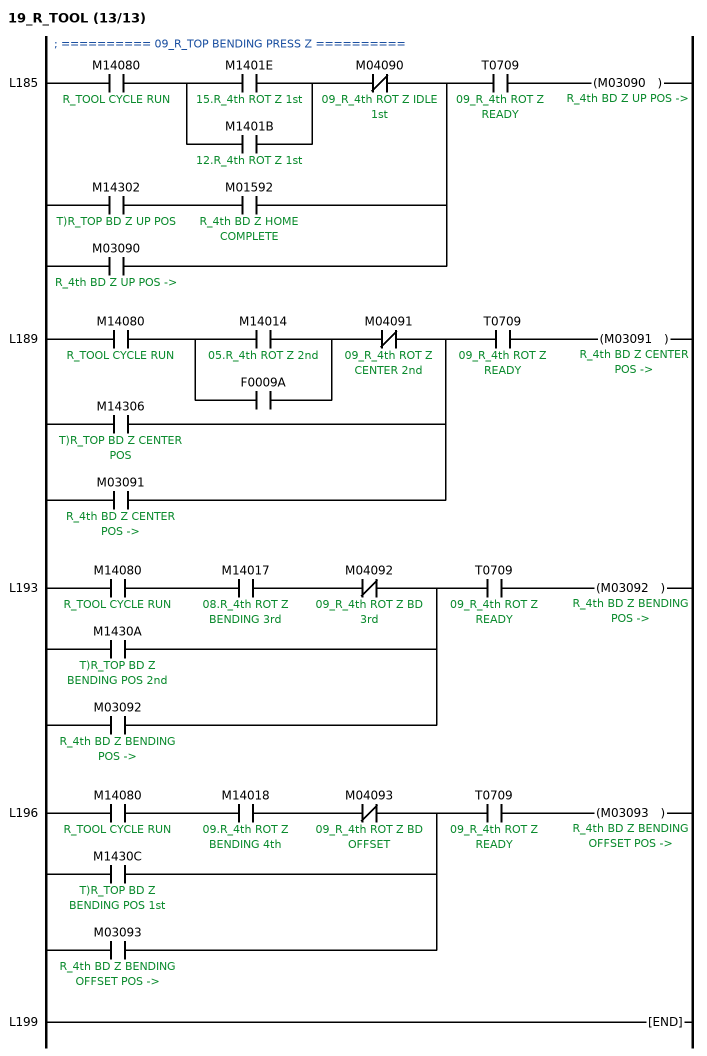
// ========== 09_R_TOP BENDING PRESS Z ==========
; L185
LOAD      M14080	// R_TOOL CYCLE RUN
LOAD      M1401E	// 15.R_4th ROT Z 1st
OR        M1401B	// 12.R_4th ROT Z 1st
AND LOAD
AND NOT   M04090	// 09_R_4th ROT Z IDLE 1st
LOAD      M14302	// T)R_TOP BD Z UP POS
AND       M01592	// R_4th BD Z HOME COMPLETE
OR LOAD
OR        M03090	// R_4th BD Z UP POS ->
AND       T0709	// 09_R_4th ROT Z READY
OUT       M03090	// R_4th BD Z UP POS ->
; L189
LOAD      M14080	// R_TOOL CYCLE RUN
LOAD      M14014	// 05.R_4th ROT Z 2nd
OR        F0009A
AND LOAD
AND NOT   M04091	// 09_R_4th ROT Z CENTER 2nd
OR        M14306	// T)R_TOP BD Z CENTER POS
OR        M03091	// R_4th BD Z CENTER POS ->
AND       T0709	// 09_R_4th ROT Z READY
OUT       M03091	// R_4th BD Z CENTER POS ->
; L193
LOAD      M14080	// R_TOOL CYCLE RUN
AND       M14017	// 08.R_4th ROT Z BENDING 3rd
AND NOT   M04092	// 09_R_4th ROT Z BD 3rd
OR        M1430A	// T)R_TOP BD Z BENDING POS 2nd
OR        M03092	// R_4th BD Z BENDING POS ->
AND       T0709	// 09_R_4th ROT Z READY
OUT       M03092	// R_4th BD Z BENDING POS ->
; L196
LOAD      M14080	// R_TOOL CYCLE RUN
AND       M14018	// 09.R_4th ROT Z BENDING 4th
AND NOT   M04093	// 09_R_4th ROT Z BD OFFSET
OR        M1430C	// T)R_TOP BD Z BENDING POS 1st
OR        M03093	// R_4th BD Z BENDING OFFSET POS ->
AND       T0709	// 09_R_4th ROT Z READY
OUT       M03093	// R_4th BD Z BENDING OFFSET POS ->
; L199
END

PROGRAM 20_R_PP (task: ¨ö¨¬A¥ì CA¡¤I¡¾¡¿¡¤¡Í)

